LIN {X 0,Y 461.075,Z 418.748,A -85,B 0,C 180,E1 -7804.212,E2 -7804.212} C_VEL
LIN {X 0,Y 463.063,Z 429.068,A -85,B 0,C 180,E1 -7806.047,E2 -7806.047} C_VEL
LIN {X 0,Y 462.7,Z 442.277,A -85,B 0,C 180,E1 -7808.247,E2 -7808.247} C_VEL
LIN {X 0,Y 462.114,Z 460.279,A -85,B 0,C 180,E1 -7811.168,E2 -7811.168} C_VEL
LIN {X 0,Y 461.868,Z 470.776,A -85,B 0,C 180,E1 -7812.78,E2 -7812.78} C_VEL
LIN {X 0,Y 464.544,Z 487.091,A -85,B 0,C 180,E1 -7813.146,E2 -7813.146} C_VEL
LIN {X 0,Y 463.76,Z 579.084,A -85,B 0,C 180,E1 -7814.593,E2 -7814.593} C_VEL
LIN {X 0,Y 463.497,Z 592.115,A -85,B 0,C 180,E1 -7814.95,E2 -7814.95} C_VEL
LIN {X 0,Y 463.114,Z 604.111,A -85,B 0,C 180,E1 -7815.443,E2 -7815.443} C_VEL
LIN {X 0,Y 462.695,Z 614.977,A -85,B 0,C 180,E1 -7816.047,E2 -7816.047} C_VEL
LIN {X 0,Y 462.205,Z 627.162,A -85,B 0,C 180,E1 -7816.928,E2 -7816.928} C_VEL
LIN {X 0,Y 461.739,Z 636.874,A -85,B 0,C 180,E1 -7817.808,E2 -7817.808} C_VEL
LIN {X 0,Y 461.187,Z 645.853,A -85,B 0,C 180,E1 -7818.796,E2 -7818.796} C_VEL
LIN {X 0,Y 460.72,Z 655.499,A -85,B 0,C 180,E1 -7820.118,E2 -7820.118} C_VEL
LIN {X 0,Y 460.302,Z 663.256,A -85,B 0,C 180,E1 -7821.439,E2 -7821.439} C_VEL
LIN {X 0,Y 460.049,Z 668.5,A -85,B 0,C 180,E1 -7822.539,E2 -7822.539} C_VEL
LIN {X 0,Y 459.926,Z 673.622,A -85,B 0,C 180,E1 -7823.86,E2 -7823.86} C_VEL
LIN {X 0,Y 459.667,Z 677.595,A -85,B 0,C 180,E1 -7825.176,E2 -7825.176} C_VEL
LIN {X 0,Y 459.685,Z 680.521,A -85,B 0,C 180,E1 -7826.494,E2 -7826.494} C_VEL
LIN {X 0,Y 459.607,Z 681.946,A -85,B 0,C 180,E1 -7827.371,E2 -7827.371} C_VEL
LIN {X 0,Y 459.523,Z 683.559,A -85,B 0,C 180,E1 -7829.124,E2 -7829.124} C_VEL
LIN {X 0,Y 459.53,Z 683.796,A -85,B 0,C 180,E1 -7830,E2 -7830} C_VEL
LIN {X 0,Y 459.523,Z 683.608,A -85,B 0,C 180,E1 -7830.876,E2 -7830.876} C_VEL
LIN {X 0,Y 459.608,Z 682.058,A -85,B 0,C 180,E1 -7832.629,E2 -7832.629} C_VEL
LIN {X 0,Y 459.685,Z 680.697,A -85,B 0,C 180,E1 -7833.506,E2 -7833.506} C_VEL
LIN {X 0,Y 459.666,Z 677.835,A -85,B 0,C 180,E1 -7834.824,E2 -7834.824} C_VEL
LIN {X 0,Y 459.903,Z 673.941,A -85,B 0,C 180,E1 -7836.141,E2 -7836.141} C_VEL
LIN {X 0,Y 460.048,Z 668.901,A -85,B 0,C 180,E1 -7837.461,E2 -7837.461} C_VEL
LIN {X 0,Y 460.356,Z 662.544,A -85,B 0,C 180,E1 -7838.781,E2 -7838.781} C_VEL
LIN {X 0,Y 460.728,Z 654.648,A -85,B 0,C 180,E1 -7840.103,E2 -7840.103} C_VEL
LIN {X 0,Y 461.174,Z 646.581,A -85,B 0,C 180,E1 -7841.204,E2 -7841.204} C_VEL
LIN {X 0,Y 461.77,Z 636.675,A -85,B 0,C 180,E1 -7842.303,E2 -7842.303} C_VEL
LIN {X 0,Y 462.278,Z 625.413,A -85,B 0,C 180,E1 -7843.305,E2 -7843.305} C_VEL
LIN {X 0,Y 462.731,Z 614.667,A -85,B 0,C 180,E1 -7844.064,E2 -7844.064} C_VEL
LIN {X 0,Y 463.159,Z 602.475,A -85,B 0,C 180,E1 -7844.724,E2 -7844.724} C_VEL
LIN {X 0,Y 463.588,Z 589.016,A -85,B 0,C 180,E1 -7845.244,E2 -7845.244} C_VEL
LIN {X 0,Y 463.856,Z 576.705,A -85,B 0,C 180,E1 -7845.545,E2 -7845.545} C_VEL
LIN {X 0,Y 464.475,Z 486.012,A -85,B 0,C 180,E1 -7846.966,E2 -7846.966} C_VEL
LIN {X 0,Y 461.849,Z 470.717,A -85,B 0,C 180,E1 -7847.319,E2 -7847.319} C_VEL
LIN {X 0,Y 462.268,Z 455.006,A -85,B 0,C 180,E1 -7849.772,E2 -7849.772} C_VEL
LIN {X 0,Y 462.866,Z 438.129,A -85,B 0,C 180,E1 -7852.544,E2 -7852.544} C_VEL
LIN {X 0,Y 463.124,Z 429.695,A -85,B 0,C 180,E1 -7853.95,E2 -7853.95} C_VEL
LIN {X 0,Y 461.038,Z 418.49,A -85,B 0,C 180,E1 -7855.922,E2 -7855.922} C_VEL
LIN {X 0,Y 460.533,Z 416.122,A -85,B 0,C 180,E1 -7856.389,E2 -7856.389} C_VEL
LIN {X 0,Y 460.519,Z 416.123,A -85,B 0,C 180,E1 -7859.555,E2 -7859.555} C_VEL
LIN {X 0,Y 460.534,Z 416.119,A -85,B 0,C 180,E1 -7862.284,E2 -7862.284} C_VEL
LIN {X 0,Y 460.511,Z 416.125,A -85,B 0,C 180,E1 -7865.446,E2 -7865.446} C_VEL
LIN {X 0,Y 460.543,Z 416.118,A -85,B 0,C 180,E1 -7868.897,E2 -7868.897} C_VEL
LIN {X 0,Y 460.526,Z 416.118,A -85,B 0,C 180,E1 -7872.181,E2 -7872.181} C_VEL
LIN {X 0,Y 460.523,Z 416.122,A -85,B 0,C 180,E1 -7875.412,E2 -7875.412} C_VEL
LIN {X 0,Y 460.535,Z 416.113,A -85,B 0,C 180,E1 -7878.397,E2 -7878.397} C_VEL
LIN {X 0,Y 460.528,Z 416.118,A -85,B 0,C 180,E1 -7881.267,E2 -7881.267} C_VEL
LIN {X 0,Y 460.511,Z 416.116,A -85,B 0,C 180,E1 -7884.554,E2 -7884.554} C_VEL
LIN {X 0,Y 460.534,Z 416.116,A -85,B 0,C 180,E1 -7887.716,E2 -7887.716} C_VEL
LIN {X 0,Y 460.523,Z 416.122,A -85,B 0,C 180,E1 -7890.768,E2 -7890.768} C_VEL
LIN {X 0,Y 460.537,Z 416.17,A -85,B 0,C 180,E1 -7893.796,E2 -7893.796} C_VEL
LIN {X 0,Y 463.051,Z 429.137,A -85,B 0,C 180,E1 -7896.046,E2 -7896.046} C_VEL
LIN {X 0,Y 462.871,Z 439.211,A -85,B 0,C 180,E1 -7897.692,E2 -7897.692} C_VEL
LIN {X 0,Y 462.206,Z 460.623,A -85,B 0,C 180,E1 -7901.159,E2 -7901.159} C_VEL
LIN {X 0,Y 461.846,Z 471.213,A -85,B 0,C 180,E1 -7902.866,E2 -7902.866} C_VEL
LIN {X 0,Y 464.307,Z 486.198,A -85,B 0,C 180,E1 -7903.224,E2 -7903.224} C_VEL
LIN {X 0,Y 463.246,Z 581.333,A -85,B 0,C 180,E1 -7904.885,E2 -7904.885} C_VEL
LIN {X 0,Y 462.876,Z 595.262,A -85,B 0,C 180,E1 -7905.323,E2 -7905.323} C_VEL
LIN {X 0,Y 462.521,Z 607.291,A -85,B 0,C 180,E1 -7905.873,E2 -7905.873} C_VEL
LIN {X 0,Y 462.061,Z 619.024,A -85,B 0,C 180,E1 -7906.588,E2 -7906.588} C_VEL
LIN {X 0,Y 461.705,Z 630.854,A -85,B 0,C 180,E1 -7907.512,E2 -7907.512} C_VEL
LIN {X 0,Y 461.134,Z 641.61,A -85,B 0,C 180,E1 -7908.572,E2 -7908.572} C_VEL
LIN {X 0,Y 460.784,Z 650.701,A -85,B 0,C 180,E1 -7909.676,E2 -7909.676} C_VEL
LIN {X 0,Y 460.359,Z 659.464,A -85,B 0,C 180,E1 -7910.997,E2 -7910.997} C_VEL
LIN {X 0,Y 460.018,Z 666.532,A -85,B 0,C 180,E1 -7912.318,E2 -7912.318} C_VEL
LIN {X 0,Y 459.857,Z 671.279,A -85,B 0,C 180,E1 -7913.414,E2 -7913.414} C_VEL
LIN {X 0,Y 459.743,Z 675.889,A -85,B 0,C 180,E1 -7914.737,E2 -7914.737} C_VEL
LIN {X 0,Y 459.644,Z 678.306,A -85,B 0,C 180,E1 -7915.615,E2 -7915.615} C_VEL
LIN {X 0,Y 459.68,Z 680.256,A -85,B 0,C 180,E1 -7916.494,E2 -7916.494} C_VEL
LIN {X 0,Y 459.607,Z 681.795,A -85,B 0,C 180,E1 -7917.371,E2 -7917.371} C_VEL
LIN {X 0,Y 459.546,Z 682.865,A -85,B 0,C 180,E1 -7918.247,E2 -7918.247} C_VEL
LIN {X 0,Y 459.53,Z 683.801,A -85,B 0,C 180,E1 -7920,E2 -7920} C_VEL
LIN {X 0,Y 459.523,Z 683.624,A -85,B 0,C 180,E1 -7920.876,E2 -7920.876} C_VEL
LIN {X 0,Y 459.607,Z 682.049,A -85,B 0,C 180,E1 -7922.629,E2 -7922.629} C_VEL
LIN {X 0,Y 459.68,Z 680.61,A -85,B 0,C 180,E1 -7923.506,E2 -7923.506} C_VEL
LIN {X 0,Y 459.657,Z 677.632,A -85,B 0,C 180,E1 -7924.824,E2 -7924.824} C_VEL
LIN {X 0,Y 459.863,Z 673.568,A -85,B 0,C 180,E1 -7926.141,E2 -7926.141} C_VEL
LIN {X 0,Y 460.032,Z 667.335,A -85,B 0,C 180,E1 -7927.682,E2 -7927.682} C_VEL
LIN {X 0,Y 460.346,Z 660.433,A -85,B 0,C 180,E1 -7929.003,E2 -7929.003} C_VEL
LIN {X 0,Y 460.752,Z 651.823,A -85,B 0,C 180,E1 -7930.325,E2 -7930.325} C_VEL
LIN {X 0,Y 461.144,Z 642.972,A -85,B 0,C 180,E1 -7931.427,E2 -7931.427} C_VEL
LIN {X 0,Y 461.659,Z 632.544,A -85,B 0,C 180,E1 -7932.479,E2 -7932.479} C_VEL
LIN {X 0,Y 462.086,Z 621.018,A -85,B 0,C 180,E1 -7933.411,E2 -7933.411} C_VEL
LIN {X 0,Y 462.511,Z 608.682,A -85,B 0,C 180,E1 -7934.183,E2 -7934.183} C_VEL
LIN {X 0,Y 462.944,Z 597.112,A -85,B 0,C 180,E1 -7934.731,E2 -7934.731} C_VEL
LIN {X 0,Y 463.231,Z 583.9,A -85,B 0,C 180,E1 -7935.172,E2 -7935.172} C_VEL
LIN {X 0,Y 463.519,Z 567.35,A -85,B 0,C 180,E1 -7935.5,E2 -7935.5} C_VEL
LIN {X 0,Y 464.548,Z 486.066,A -85,B 0,C 180,E1 -7936.986,E2 -7936.986} C_VEL
LIN {X 0,Y 462.152,Z 471.916,A -85,B 0,C 180,E1 -7937.398,E2 -7937.398} C_VEL
LIN {X 0,Y 462.715,Z 452.676,A -85,B 0,C 180,E1 -7940.447,E2 -7940.447} C_VEL
LIN {X 0,Y 463.248,Z 433.335,A -85,B 0,C 180,E1 -7943.468,E2 -7943.468} C_VEL
LIN {X 0,Y 463.221,Z 428.858,A -85,B 0,C 180,E1 -7944.183,E2 -7944.183} C_VEL
LIN {X 0,Y 461.093,Z 418.517,A -85,B 0,C 180,E1 -7945.936,E2 -7945.936} C_VEL
LIN {X 0,Y 460.518,Z 416.124,A -85,B 0,C 180,E1 -7946.36,E2 -7946.36} C_VEL
LIN {X 0,Y 460.519,Z 416.126,A -85,B 0,C 180,E1 -7949.555,E2 -7949.555} C_VEL
LIN {X 0,Y 460.533,Z 416.119,A -85,B 0,C 180,E1 -7952.284,E2 -7952.284} C_VEL
LIN {X 0,Y 460.511,Z 416.125,A -85,B 0,C 180,E1 -7955.446,E2 -7955.446} C_VEL
LIN {X 0,Y 460.546,Z 416.118,A -85,B 0,C 180,E1 -7958.897,E2 -7958.897} C_VEL
LIN {X 0,Y 460.525,Z 416.118,A -85,B 0,C 180,E1 -7962.181,E2 -7962.181} C_VEL
LIN {X 0,Y 460.52,Z 416.122,A -85,B 0,C 180,E1 -7965.411,E2 -7965.411} C_VEL
LIN {X 0,Y 460.534,Z 416.12,A -85,B 0,C 180,E1 -7968.397,E2 -7968.397} C_VEL
LIN {X 0,Y 460.527,Z 416.119,A -85,B 0,C 180,E1 -7971.267,E2 -7971.267} C_VEL
LIN {X 0,Y 460.511,Z 416.122,A -85,B 0,C 180,E1 -7974.554,E2 -7974.554} C_VEL
LIN {X 0,Y 460.533,Z 416.118,A -85,B 0,C 180,E1 -7977.716,E2 -7977.716} C_VEL
LIN {X 0,Y 460.546,Z 416.195,A -85,B 0,C 180,E1 -7981.019,E2 -7981.019} C_VEL
LIN {X 0,Y 463.789,Z 431.549,A -85,B 0,C 180,E1 -7983.587,E2 -7983.587} C_VEL
LIN {X 0,Y 463.673,Z 438.411,A -85,B 0,C 180,E1 -7984.647,E2 -7984.647} C_VEL
LIN {X 0,Y 462.791,Z 458.476,A -85,B 0,C 180,E1 -7987.688,E2 -7987.688} C_VEL
LIN {X 0,Y 461.825,Z 481.82,A -85,B 0,C 180,E1 -7991.173,E2 -7991.173} C_VEL
LIN {X 0,Y 461.381,Z 492.48,A -85,B 0,C 180,E1 -7992.75,E2 -7992.75} C_VEL
LIN {X 0,Y 464.124,Z 514.756,A -85,B 0,C 180,E1 -7993.251,E2 -7993.251} C_VEL
LIN {X 0,Y 463.33,Z 592.644,A -85,B 0,C 180,E1 -7994.578,E2 -7994.578} C_VEL
LIN {X 0,Y 463.11,Z 609.106,A -85,B 0,C 180,E1 -7994.881,E2 -7994.881} C_VEL
LIN {X 0,Y 462.775,Z 621.21,A -85,B 0,C 180,E1 -7995.263,E2 -7995.263} C_VEL
LIN {X 0,Y 462.308,Z 633.167,A -85,B 0,C 180,E1 -7995.81,E2 -7995.81} C_VEL
LIN {X 0,Y 461.887,Z 645.584,A -85,B 0,C 180,E1 -7996.583,E2 -7996.583} C_VEL
LIN {X 0,Y 461.421,Z 656.045,A -85,B 0,C 180,E1 -7997.412,E2 -7997.412} C_VEL
LIN {X 0,Y 460.979,Z 665.561,A -85,B 0,C 180,E1 -7998.346,E2 -7998.346} C_VEL
LIN {X 0,Y 460.53,Z 674.702,A -85,B 0,C 180,E1 -7999.448,E2 -7999.448} C_VEL
LIN {X 0,Y 460.165,Z 683.581,A -85,B 0,C 180,E1 -8000.772,E2 -8000.772} C_VEL
LIN {X 0,Y 459.921,Z 690.697,A -85,B 0,C 180,E1 -8002.095,E2 -8002.095} C_VEL
LIN {X 0,Y 459.719,Z 696.887,A -85,B 0,C 180,E1 -8003.564,E2 -8003.564} C_VEL
LIN {X 0,Y 459.652,Z 702.015,A -85,B 0,C 180,E1 -8005.176,E2 -8005.176} C_VEL
LIN {X 0,Y 459.697,Z 704.999,A -85,B 0,C 180,E1 -8006.494,E2 -8006.494} C_VEL
LIN {X 0,Y 459.64,Z 706.431,A -85,B 0,C 180,E1 -8007.371,E2 -8007.371} C_VEL
LIN {X 0,Y 459.596,Z 708.057,A -85,B 0,C 180,E1 -8009.124,E2 -8009.124} C_VEL
LIN {X 0,Y 459.584,Z 708.278,A -85,B 0,C 180,E1 -8010,E2 -8010} C_VEL
LIN {X 0,Y 459.596,Z 708.057,A -85,B 0,C 180,E1 -8010.876,E2 -8010.876} C_VEL
LIN {X 0,Y 459.642,Z 706.431,A -85,B 0,C 180,E1 -8012.629,E2 -8012.629} C_VEL
LIN {X 0,Y 459.708,Z 705,A -85,B 0,C 180,E1 -8013.506,E2 -8013.506} C_VEL
LIN {X 0,Y 459.66,Z 702.015,A -85,B 0,C 180,E1 -8014.824,E2 -8014.824} C_VEL
LIN {X 0,Y 459.765,Z 696.7,A -85,B 0,C 180,E1 -8016.487,E2 -8016.487} C_VEL
LIN {X 0,Y 459.925,Z 690.699,A -85,B 0,C 180,E1 -8017.905,E2 -8017.905} C_VEL
LIN {X 0,Y 460.19,Z 683.584,A -85,B 0,C 180,E1 -8019.228,E2 -8019.228} C_VEL
LIN {X 0,Y 460.54,Z 674.691,A -85,B 0,C 180,E1 -8020.552,E2 -8020.552} C_VEL
LIN {X 0,Y 460.979,Z 665.542,A -85,B 0,C 180,E1 -8021.654,E2 -8021.654} C_VEL
LIN {X 0,Y 461.492,Z 655.22,A -85,B 0,C 180,E1 -8022.656,E2 -8022.656} C_VEL
LIN {X 0,Y 461.929,Z 643.989,A -85,B 0,C 180,E1 -8023.528,E2 -8023.528} C_VEL
LIN {X 0,Y 462.4,Z 632.124,A -85,B 0,C 180,E1 -8024.243,E2 -8024.243} C_VEL
LIN {X 0,Y 462.835,Z 619.661,A -85,B 0,C 180,E1 -8024.791,E2 -8024.791} C_VEL
LIN {X 0,Y 463.161,Z 606.804,A -85,B 0,C 180,E1 -8025.174,E2 -8025.174} C_VEL
LIN {X 0,Y 463.762,Z 546.734,A -85,B 0,C 180,E1 -8026.193,E2 -8026.193} C_VEL
LIN {X 0,Y 464.092,Z 513.352,A -85,B 0,C 180,E1 -8026.813,E2 -8026.813} C_VEL
LIN {X 0,Y 461.241,Z 488.658,A -85,B 0,C 180,E1 -8027.437,E2 -8027.437} C_VEL
LIN {X 0,Y 462.12,Z 465.23,A -85,B 0,C 180,E1 -8030.94,E2 -8030.94} C_VEL
LIN {X 0,Y 463.02,Z 444.03,A -85,B 0,C 180,E1 -8034.194,E2 -8034.194} C_VEL
LIN {X 0,Y 463.674,Z 432.077,A -85,B 0,C 180,E1 -8036.076,E2 -8036.076} C_VEL
LIN {X 0,Y 462.51,Z 424.778,A -85,B 0,C 180,E1 -8037.341,E2 -8037.341} C_VEL
LIN {X 0,Y 460.541,Z 416.122,A -85,B 0,C 180,E1 -8038.981,E2 -8038.981} C_VEL
LIN {X 0,Y 460.533,Z 416.12,A -85,B 0,C 180,E1 -8042.284,E2 -8042.284} C_VEL
LIN {X 0,Y 460.51,Z 416.125,A -85,B 0,C 180,E1 -8045.446,E2 -8045.446} C_VEL
LIN {X 0,Y 460.534,Z 416.119,A -85,B 0,C 180,E1 -8048.896,E2 -8048.896} C_VEL
LIN {X 0,Y 460.52,Z 416.122,A -85,B 0,C 180,E1 -8051.601,E2 -8051.601} C_VEL
LIN {X 0,Y 460.518,Z 416.12,A -85,B 0,C 180,E1 -8054.589,E2 -8054.589} C_VEL
LIN {X 0,Y 460.525,Z 416.118,A -85,B 0,C 180,E1 -8057.819,E2 -8057.819} C_VEL
LIN {X 0,Y 460.547,Z 416.119,A -85,B 0,C 180,E1 -8061.102,E2 -8061.102} C_VEL
LIN {X 0,Y 460.513,Z 416.121,A -85,B 0,C 180,E1 -8064.554,E2 -8064.554} C_VEL
LIN {X 0,Y 460.534,Z 416.118,A -85,B 0,C 180,E1 -8067.716,E2 -8067.716} C_VEL
LIN {X 0,Y 460.542,Z 416.121,A -85,B 0,C 180,E1 -8070.769,E2 -8070.769} C_VEL
LIN {X 0,Y 460.559,Z 416.116,A -85,B 0,C 180,E1 -8073.734,E2 -8073.734} C_VEL
LIN {X 0,Y 460.547,Z 416.123,A -85,B 0,C 180,E1 -8076.624,E2 -8076.624} C_VEL
LIN {X 0,Y 460.553,Z 416.117,A -85,B 0,C 180,E1 -8079.453,E2 -8079.453} C_VEL
LIN {X 0,Y 460.568,Z 416.117,A -85,B 0,C 180,E1 -8082.643,E2 -8082.643} C_VEL
LIN {X 0,Y 460.578,Z 416.182,A -85,B 0,C 180,E1 -8082.713,E2 -8082.713} C_VEL
LIN {X 0,Y 462.882,Z 422.42,A -85,B 0,C 180,E1 -8082.954,E2 -8082.954} C_VEL
LIN {X 0,Y 464.811,Z 427.449,A -85,B 0,C 180,E1 -8083.149,E2 -8083.149} C_VEL
LIN {X 0,Y 463.534,Z 519.172,A -85,B 0,C 180,E1 -8084.867,E2 -8084.867} C_VEL
LIN {X 0,Y 463.331,Z 532.093,A -85,B 0,C 180,E1 -8085.281,E2 -8085.281} C_VEL
LIN {X 0,Y 463.084,Z 544.075,A -85,B 0,C 180,E1 -8085.835,E2 -8085.835} C_VEL
LIN {X 0,Y 462.679,Z 555.95,A -85,B 0,C 180,E1 -8086.568,E2 -8086.568} C_VEL
LIN {X 0,Y 462.241,Z 567.55,A -85,B 0,C 180,E1 -8087.487,E2 -8087.487} C_VEL
LIN {X 0,Y 461.85,Z 576.525,A -85,B 0,C 180,E1 -8088.368,E2 -8088.368} C_VEL
LIN {X 0,Y 461.424,Z 585.721,A -85,B 0,C 180,E1 -8089.469,E2 -8089.469} C_VEL
LIN {X 0,Y 460.993,Z 594.604,A -85,B 0,C 180,E1 -8090.789,E2 -8090.789} C_VEL
LIN {X 0,Y 460.65,Z 601.715,A -85,B 0,C 180,E1 -8092.108,E2 -8092.108} C_VEL
LIN {X 0,Y 460.422,Z 607.329,A -85,B 0,C 180,E1 -8093.426,E2 -8093.426} C_VEL
LIN {X 0,Y 460.148,Z 611.72,A -85,B 0,C 180,E1 -8094.742,E2 -8094.742} C_VEL
LIN {X 0,Y 460.171,Z 614,A -85,B 0,C 180,E1 -8095.62,E2 -8095.62} C_VEL
LIN {X 0,Y 459.993,Z 615.87,A -85,B 0,C 180,E1 -8096.496,E2 -8096.496} C_VEL
LIN {X 0,Y 459.819,Z 617.29,A -85,B 0,C 180,E1 -8097.372,E2 -8097.372} C_VEL
LIN {X 0,Y 459.691,Z 618.83,A -85,B 0,C 180,E1 -8099.124,E2 -8099.124} C_VEL
LIN {X 0,Y 459.679,Z 619.005,A -85,B 0,C 180,E1 -8100,E2 -8100} C_VEL
LIN {X 0,Y 459.679,Z 618.737,A -85,B 0,C 180,E1 -8100.876,E2 -8100.876} C_VEL
LIN {X 0,Y 459.806,Z 616.987,A -85,B 0,C 180,E1 -8102.628,E2 -8102.628} C_VEL
LIN {X 0,Y 459.987,Z 615.491,A -85,B 0,C 180,E1 -8103.504,E2 -8103.504} C_VEL
LIN {X 0,Y 460.064,Z 612.422,A -85,B 0,C 180,E1 -8104.82,E2 -8104.82} C_VEL
LIN {X 0,Y 460.201,Z 607.217,A -85,B 0,C 180,E1 -8106.421,E2 -8106.421} C_VEL
LIN {X 0,Y 460.446,Z 600.884,A -85,B 0,C 180,E1 -8107.896,E2 -8107.896} C_VEL
LIN {X 0,Y 460.798,Z 593.657,A -85,B 0,C 180,E1 -8109.215,E2 -8109.215} C_VEL
LIN {X 0,Y 461.192,Z 584.638,A -85,B 0,C 180,E1 -8110.537,E2 -8110.537} C_VEL
LIN {X 0,Y 461.645,Z 575.368,A -85,B 0,C 180,E1 -8111.637,E2 -8111.637} C_VEL
LIN {X 0,Y 462.056,Z 565.037,A -85,B 0,C 180,E1 -8112.63,E2 -8112.63} C_VEL
LIN {X 0,Y 462.46,Z 553.768,A -85,B 0,C 180,E1 -8113.499,E2 -8113.499} C_VEL
LIN {X 0,Y 462.783,Z 541.687,A -85,B 0,C 180,E1 -8114.231,E2 -8114.231} C_VEL
LIN {X 0,Y 463.115,Z 528.597,A -85,B 0,C 180,E1 -8114.81,E2 -8114.81} C_VEL
LIN {X 0,Y 463.364,Z 515.877,A -85,B 0,C 180,E1 -8115.195,E2 -8115.195} C_VEL
LIN {X 0,Y 464.244,Z 426.98,A -85,B 0,C 180,E1 -8116.76,E2 -8116.76} C_VEL
LIN {X 0,Y 460.544,Z 416.12,A -85,B 0,C 180,E1 -8117.112,E2 -8117.112} C_VEL
LIN {X 0,Y 460.569,Z 416.121,A -85,B 0,C 180,E1 -8119.616,E2 -8119.616} C_VEL
LIN {X 0,Y 460.513,Z 416.117,A -85,B 0,C 180,E1 -8122.429,E2 -8122.429} C_VEL
LIN {X 0,Y 460.548,Z 416.115,A -85,B 0,C 180,E1 -8125.796,E2 -8125.796} C_VEL
LIN {X 0,Y 460.552,Z 416.11,A -85,B 0,C 180,E1 -8128.233,E2 -8128.233} C_VEL
LIN {X 0,Y 460.524,Z 416.118,A -85,B 0,C 180,E1 -8131.283,E2 -8131.283} C_VEL
LIN {X 0,Y 460.534,Z 416.105,A -85,B 0,C 180,E1 -8134.505,E2 -8134.505} C_VEL
LIN {X 0,Y 460.504,Z 416.122,A -85,B 0,C 180,E1 -8137.623,E2 -8137.623} C_VEL
LIN {X 0,Y 460.542,Z 416.109,A -85,B 0,C 180,E1 -8140.269,E2 -8140.269} C_VEL
LIN {X 0,Y 460.503,Z 416.123,A -85,B 0,C 180,E1 -8143.375,E2 -8143.375} C_VEL
LIN {X 0,Y 460.503,Z 416.118,A -85,B 0,C 180,E1 -8146.625,E2 -8146.625} C_VEL
LIN {X 0,Y 460.542,Z 416.11,A -85,B 0,C 180,E1 -8149.731,E2 -8149.731} C_VEL
LIN {X 0,Y 460.499,Z 416.124,A -85,B 0,C 180,E1 -8152.524,E2 -8152.524} C_VEL
LIN {X 0,Y 460.548,Z 416.114,A -85,B 0,C 180,E1 -8155.624,E2 -8155.624} C_VEL
LIN {X 0,Y 460.54,Z 416.122,A -85,B 0,C 180,E1 -8158.745,E2 -8158.745} C_VEL
LIN {X 0,Y 460.51,Z 416.125,A -85,B 0,C 180,E1 -8161.764,E2 -8161.764} C_VEL
LIN {X 0,Y 460.555,Z 416.234,A -85,B 0,C 180,E1 -8163.765,E2 -8163.765} C_VEL
LIN {X 0,Y 461.075,Z 418.748,A -85,B 0,C 180,E1 -8164.212,E2 -8164.212} C_VEL
LIN {X 0,Y 461.098,Z 422.256,A -85,B 0,C 180,E1 -8164.803,E2 -8164.803} C_VEL
LIN {X 0,Y 460.118,Z 425.937,A -85,B 0,C 180,E1 -8165.373,E2 -8165.373} C_VEL
LIN {X 0,Y 456.381,Z 435.933,A -85,B 0,C 180,E1 -8166.877,E2 -8166.877} C_VEL
LIN {X 0,Y 455.999,Z 438.386,A -85,B 0,C 180,E1 -8167.274,E2 -8167.274} C_VEL
LIN {X 0,Y 455.271,Z 457.786,A -85,B 0,C 180,E1 -8170.476,E2 -8170.476} C_VEL
LIN {X 0,Y 454.939,Z 470.902,A -85,B 0,C 180,E1 -8172.51,E2 -8172.51} C_VEL
LIN {X 0,Y 457.737,Z 487.036,A -85,B 0,C 180,E1 -8172.885,E2 -8172.885} C_VEL
LIN {X 0,Y 456.936,Z 579.198,A -85,B 0,C 180,E1 -8174.357,E2 -8174.357} C_VEL
LIN {X 0,Y 456.665,Z 592.262,A -85,B 0,C 180,E1 -8174.719,E2 -8174.719} C_VEL
LIN {X 0,Y 456.271,Z 604.275,A -85,B 0,C 180,E1 -8175.22,E2 -8175.22} C_VEL
LIN {X 0,Y 455.814,Z 615.149,A -85,B 0,C 180,E1 -8175.832,E2 -8175.832} C_VEL
LIN {X 0,Y 455.286,Z 627.235,A -85,B 0,C 180,E1 -8176.717,E2 -8176.717} C_VEL
LIN {X 0,Y 454.82,Z 637.055,A -85,B 0,C 180,E1 -8177.62,E2 -8177.62} C_VEL
LIN {X 0,Y 454.232,Z 646.036,A -85,B 0,C 180,E1 -8178.623,E2 -8178.623} C_VEL
LIN {X 0,Y 453.768,Z 654.242,A -85,B 0,C 180,E1 -8179.74,E2 -8179.74} C_VEL
LIN {X 0,Y 453.355,Z 662.245,A -85,B 0,C 180,E1 -8181.082,E2 -8181.082} C_VEL
LIN {X 0,Y 452.992,Z 668.688,A -85,B 0,C 180,E1 -8182.422,E2 -8182.422} C_VEL
LIN {X 0,Y 452.856,Z 673.811,A -85,B 0,C 180,E1 -8183.763,E2 -8183.763} C_VEL
LIN {X 0,Y 452.6,Z 677.784,A -85,B 0,C 180,E1 -8185.101,E2 -8185.101} C_VEL
LIN {X 0,Y 452.601,Z 680.711,A -85,B 0,C 180,E1 -8186.439,E2 -8186.439} C_VEL
LIN {X 0,Y 452.534,Z 682.135,A -85,B 0,C 180,E1 -8187.33,E2 -8187.33} C_VEL
LIN {X 0,Y 452.43,Z 683.748,A -85,B 0,C 180,E1 -8189.11,E2 -8189.11} C_VEL
LIN {X 0,Y 452.435,Z 683.985,A -85,B 0,C 180,E1 -8190,E2 -8190} C_VEL
LIN {X 0,Y 452.43,Z 683.796,A -85,B 0,C 180,E1 -8190.89,E2 -8190.89} C_VEL
LIN {X 0,Y 452.534,Z 682.246,A -85,B 0,C 180,E1 -8192.67,E2 -8192.67} C_VEL
LIN {X 0,Y 452.601,Z 680.884,A -85,B 0,C 180,E1 -8193.561,E2 -8193.561} C_VEL
LIN {X 0,Y 452.599,Z 678.022,A -85,B 0,C 180,E1 -8194.899,E2 -8194.899} C_VEL
LIN {X 0,Y 452.831,Z 674.127,A -85,B 0,C 180,E1 -8196.237,E2 -8196.237} C_VEL
LIN {X 0,Y 452.991,Z 669.086,A -85,B 0,C 180,E1 -8197.578,E2 -8197.578} C_VEL
LIN {X 0,Y 453.34,Z 662.726,A -85,B 0,C 180,E1 -8198.918,E2 -8198.918} C_VEL
LIN {X 0,Y 453.739,Z 654.828,A -85,B 0,C 180,E1 -8200.261,E2 -8200.261} C_VEL
LIN {X 0,Y 454.21,Z 646.758,A -85,B 0,C 180,E1 -8201.378,E2 -8201.378} C_VEL
LIN {X 0,Y 454.835,Z 636.848,A -85,B 0,C 180,E1 -8202.493,E2 -8202.493} C_VEL
LIN {X 0,Y 455.346,Z 625.724,A -85,B 0,C 180,E1 -8203.499,E2 -8203.499} C_VEL
LIN {X 0,Y 455.851,Z 614.825,A -85,B 0,C 180,E1 -8204.281,E2 -8204.281} C_VEL
LIN {X 0,Y 456.318,Z 602.616,A -85,B 0,C 180,E1 -8204.95,E2 -8204.95} C_VEL
LIN {X 0,Y 456.761,Z 589.133,A -85,B 0,C 180,E1 -8205.478,E2 -8205.478} C_VEL
LIN {X 0,Y 457.046,Z 576.746,A -85,B 0,C 180,E1 -8205.782,E2 -8205.782} C_VEL
LIN {X 0,Y 457.62,Z 486.269,A -85,B 0,C 180,E1 -8207.224,E2 -8207.224} C_VEL
LIN {X 0,Y 454.952,Z 470.855,A -85,B 0,C 180,E1 -8207.587,E2 -8207.587} C_VEL
LIN {X 0,Y 455.382,Z 454.985,A -85,B 0,C 180,E1 -8210.084,E2 -8210.084} C_VEL
LIN {X 0,Y 456.034,Z 437.992,A -85,B 0,C 180,E1 -8212.901,E2 -8212.901} C_VEL
LIN {X 0,Y 456.194,Z 430.883,A -85,B 0,C 180,E1 -8214.091,E2 -8214.091} C_VEL
LIN {X 0,Y 453.772,Z 418.331,A -85,B 0,C 180,E1 -8216.336,E2 -8216.336} C_VEL
LIN {X 0,Y 453.472,Z 417.002,A -85,B 0,C 180,E1 -8216.62,E2 -8216.62} C_VEL
LIN {X 0,Y 453.471,Z 417.001,A -85,B 0,C 180,E1 -8219.784,E2 -8219.784} C_VEL
LIN {X 0,Y 453.493,Z 416.998,A -85,B 0,C 180,E1 -8223.189,E2 -8223.189} C_VEL
LIN {X 0,Y 453.453,Z 417.001,A -85,B 0,C 180,E1 -8226.298,E2 -8226.298} C_VEL
LIN {X 0,Y 453.488,Z 416.995,A -85,B 0,C 180,E1 -8229.45,E2 -8229.45} C_VEL
LIN {X 0,Y 453.479,Z 416.996,A -85,B 0,C 180,E1 -8231.935,E2 -8231.935} C_VEL
LIN {X 0,Y 453.494,Z 416.997,A -85,B 0,C 180,E1 -8235.47,E2 -8235.47} C_VEL
LIN {X 0,Y 453.482,Z 416.991,A -85,B 0,C 180,E1 -8238.209,E2 -8238.209} C_VEL
LIN {X 0,Y 453.512,Z 416.998,A -85,B 0,C 180,E1 -8240.791,E2 -8240.791} C_VEL
LIN {X 0,Y 453.454,Z 416.989,A -85,B 0,C 180,E1 -8243.917,E2 -8243.917} C_VEL
LIN {X 0,Y 453.486,Z 416.996,A -85,B 0,C 180,E1 -8247.151,E2 -8247.151} C_VEL
LIN {X 0,Y 453.465,Z 417.002,A -85,B 0,C 180,E1 -8250.267,E2 -8250.267} C_VEL
LIN {X 0,Y 453.492,Z 416.996,A -85,B 0,C 180,E1 -8253.574,E2 -8253.574} C_VEL
LIN {X 0,Y 456.116,Z 430.323,A -85,B 0,C 180,E1 -8255.92,E2 -8255.92} C_VEL
LIN {X 0,Y 456.042,Z 438.922,A -85,B 0,C 180,E1 -8257.339,E2 -8257.339} C_VEL
LIN {X 0,Y 455.275,Z 460.69,A -85,B 0,C 180,E1 -8260.89,E2 -8260.89} C_VEL
LIN {X 0,Y 454.879,Z 471.285,A -85,B 0,C 180,E1 -8262.614,E2 -8262.614} C_VEL
LIN {X 0,Y 457.419,Z 486.804,A -85,B 0,C 180,E1 -8262.997,E2 -8262.997} C_VEL
LIN {X 0,Y 456.349,Z 580.94,A -85,B 0,C 180,E1 -8264.68,E2 -8264.68} C_VEL
LIN {X 0,Y 455.963,Z 594.3,A -85,B 0,C 180,E1 -8265.095,E2 -8265.095} C_VEL
LIN {X 0,Y 455.613,Z 606.644,A -85,B 0,C 180,E1 -8265.654,E2 -8265.654} C_VEL
LIN {X 0,Y 455.112,Z 618.568,A -85,B 0,C 180,E1 -8266.379,E2 -8266.379} C_VEL
LIN {X 0,Y 454.817,Z 628.793,A -85,B 0,C 180,E1 -8267.169,E2 -8267.169} C_VEL
LIN {X 0,Y 454.284,Z 639.377,A -85,B 0,C 180,E1 -8268.171,E2 -8268.171} C_VEL
LIN {X 0,Y 453.787,Z 648.868,A -85,B 0,C 180,E1 -8269.289,E2 -8269.289} C_VEL
LIN {X 0,Y 453.352,Z 658.109,A -85,B 0,C 180,E1 -8270.632,E2 -8270.632} C_VEL
LIN {X 0,Y 453.022,Z 665.453,A -85,B 0,C 180,E1 -8271.974,E2 -8271.974} C_VEL
LIN {X 0,Y 452.769,Z 671.8,A -85,B 0,C 180,E1 -8273.428,E2 -8273.428} C_VEL
LIN {X 0,Y 452.688,Z 675.981,A -85,B 0,C 180,E1 -8274.655,E2 -8274.655} C_VEL
LIN {X 0,Y 452.558,Z 678.427,A -85,B 0,C 180,E1 -8275.547,E2 -8275.547} C_VEL
LIN {X 0,Y 452.581,Z 680.393,A -85,B 0,C 180,E1 -8276.439,E2 -8276.439} C_VEL
LIN {X 0,Y 452.533,Z 681.947,A -85,B 0,C 180,E1 -8277.33,E2 -8277.33} C_VEL
LIN {X 0,Y 452.461,Z 683.036,A -85,B 0,C 180,E1 -8278.22,E2 -8278.22} C_VEL
LIN {X 0,Y 452.435,Z 683.991,A -85,B 0,C 180,E1 -8280,E2 -8280} C_VEL
LIN {X 0,Y 452.43,Z 683.826,A -85,B 0,C 180,E1 -8280.89,E2 -8280.89} C_VEL
LIN {X 0,Y 452.461,Z 683.241,A -85,B 0,C 180,E1 -8281.78,E2 -8281.78} C_VEL
LIN {X 0,Y 452.533,Z 682.259,A -85,B 0,C 180,E1 -8282.67,E2 -8282.67} C_VEL
LIN {X 0,Y 452.596,Z 680.827,A -85,B 0,C 180,E1 -8283.561,E2 -8283.561} C_VEL
LIN {X 0,Y 452.591,Z 677.847,A -85,B 0,C 180,E1 -8284.899,E2 -8284.899} C_VEL
LIN {X 0,Y 452.792,Z 673.779,A -85,B 0,C 180,E1 -8286.238,E2 -8286.238} C_VEL
LIN {X 0,Y 452.995,Z 667.544,A -85,B 0,C 180,E1 -8287.802,E2 -8287.802} C_VEL
LIN {X 0,Y 453.334,Z 660.639,A -85,B 0,C 180,E1 -8289.143,E2 -8289.143} C_VEL
LIN {X 0,Y 453.768,Z 652.028,A -85,B 0,C 180,E1 -8290.485,E2 -8290.485} C_VEL
LIN {X 0,Y 454.188,Z 643.159,A -85,B 0,C 180,E1 -8291.605,E2 -8291.605} C_VEL
LIN {X 0,Y 454.712,Z 632.916,A -85,B 0,C 180,E1 -8292.656,E2 -8292.656} C_VEL
LIN {X 0,Y 455.145,Z 622.743,A -85,B 0,C 180,E1 -8293.506,E2 -8293.506} C_VEL
LIN {X 0,Y 455.565,Z 610.878,A -85,B 0,C 180,E1 -8294.29,E2 -8294.29} C_VEL
LIN {X 0,Y 456.02,Z 598.658,A -85,B 0,C 180,E1 -8294.903,E2 -8294.903} C_VEL
LIN {X 0,Y 456.353,Z 586.282,A -85,B 0,C 180,E1 -8295.349,E2 -8295.349} C_VEL
LIN {X 0,Y 456.663,Z 571.158,A -85,B 0,C 180,E1 -8295.681,E2 -8295.681} C_VEL
LIN {X 0,Y 457.931,Z 487.484,A -85,B 0,C 180,E1 -8297.254,E2 -8297.254} C_VEL
LIN {X 0,Y 455.317,Z 472.331,A -85,B 0,C 180,E1 -8297.691,E2 -8297.691} C_VEL
LIN {X 0,Y 455.897,Z 453.053,A -85,B 0,C 180,E1 -8300.767,E2 -8300.767} C_VEL
LIN {X 0,Y 456.456,Z 435.128,A -85,B 0,C 180,E1 -8303.598,E2 -8303.598} C_VEL
LIN {X 0,Y 456.35,Z 430.149,A -85,B 0,C 180,E1 -8304.405,E2 -8304.405} C_VEL
LIN {X 0,Y 454.003,Z 419.118,A -85,B 0,C 180,E1 -8306.324,E2 -8306.324} C_VEL
LIN {X 0,Y 453.477,Z 417,A -85,B 0,C 180,E1 -8306.708,E2 -8306.708} C_VEL
LIN {X 0,Y 453.47,Z 417.004,A -85,B 0,C 180,E1 -8309.784,E2 -8309.784} C_VEL
LIN {X 0,Y 453.493,Z 417,A -85,B 0,C 180,E1 -8313.189,E2 -8313.189} C_VEL
LIN {X 0,Y 453.452,Z 416.999,A -85,B 0,C 180,E1 -8316.298,E2 -8316.298} C_VEL
LIN {X 0,Y 453.492,Z 416.996,A -85,B 0,C 180,E1 -8319.45,E2 -8319.45} C_VEL
LIN {X 0,Y 453.479,Z 416.997,A -85,B 0,C 180,E1 -8321.935,E2 -8321.935} C_VEL
LIN {X 0,Y 453.49,Z 416.998,A -85,B 0,C 180,E1 -8325.471,E2 -8325.471} C_VEL
LIN {X 0,Y 453.481,Z 416.997,A -85,B 0,C 180,E1 -8328.209,E2 -8328.209} C_VEL
LIN {X 0,Y 453.496,Z 416.995,A -85,B 0,C 180,E1 -8330.793,E2 -8330.793} C_VEL
LIN {X 0,Y 453.453,Z 416.999,A -85,B 0,C 180,E1 -8333.917,E2 -8333.917} C_VEL
LIN {X 0,Y 453.485,Z 416.997,A -85,B 0,C 180,E1 -8337.151,E2 -8337.151} C_VEL
LIN {X 0,Y 453.513,Z 416.997,A -85,B 0,C 180,E1 -8340.781,E2 -8340.781} C_VEL
LIN {X 0,Y 456.87,Z 433.019,A -85,B 0,C 180,E1 -8343.506,E2 -8343.506} C_VEL
LIN {X 0,Y 456.522,Z 445.458,A -85,B 0,C 180,E1 -8345.439,E2 -8345.439} C_VEL
LIN {X 0,Y 455.514,Z 465.486,A -85,B 0,C 180,E1 -8348.504,E2 -8348.504} C_VEL
LIN {X 0,Y 454.546,Z 488.512,A -85,B 0,C 180,E1 -8351.987,E2 -8351.987} C_VEL
LIN {X 0,Y 454.401,Z 491.955,A -85,B 0,C 180,E1 -8352.505,E2 -8352.505} C_VEL
LIN {X 0,Y 457.276,Z 516.196,A -85,B 0,C 180,E1 -8353.051,E2 -8353.051} C_VEL
LIN {X 0,Y 456.674,Z 569.237,A -85,B 0,C 180,E1 -8353.975,E2 -8353.975} C_VEL
LIN {X 0,Y 456.26,Z 606.763,A -85,B 0,C 180,E1 -8354.591,E2 -8354.591} C_VEL
LIN {X 0,Y 455.946,Z 620.322,A -85,B 0,C 180,E1 -8355.009,E2 -8355.009} C_VEL
LIN {X 0,Y 455.413,Z 633.01,A -85,B 0,C 180,E1 -8355.591,E2 -8355.591} C_VEL
LIN {X 0,Y 454.966,Z 645.418,A -85,B 0,C 180,E1 -8356.375,E2 -8356.375} C_VEL
LIN {X 0,Y 454.447,Z 656.302,A -85,B 0,C 180,E1 -8357.254,E2 -8357.254} C_VEL
LIN {X 0,Y 453.949,Z 665.383,A -85,B 0,C 180,E1 -8358.163,E2 -8358.163} C_VEL
LIN {X 0,Y 453.525,Z 674.521,A -85,B 0,C 180,E1 -8359.283,E2 -8359.283} C_VEL
LIN {X 0,Y 453.134,Z 683.398,A -85,B 0,C 180,E1 -8360.627,E2 -8360.627} C_VEL
LIN {X 0,Y 452.856,Z 690.511,A -85,B 0,C 180,E1 -8361.971,E2 -8361.971} C_VEL
LIN {X 0,Y 452.63,Z 697.132,A -85,B 0,C 180,E1 -8363.582,E2 -8363.582} C_VEL
LIN {X 0,Y 452.579,Z 701.828,A -85,B 0,C 180,E1 -8365.1,E2 -8365.1} C_VEL
LIN {X 0,Y 452.59,Z 704.811,A -85,B 0,C 180,E1 -8366.439,E2 -8366.439} C_VEL
LIN {X 0,Y 452.564,Z 706.243,A -85,B 0,C 180,E1 -8367.33,E2 -8367.33} C_VEL
LIN {X 0,Y 452.499,Z 707.868,A -85,B 0,C 180,E1 -8369.11,E2 -8369.11} C_VEL
LIN {X 0,Y 452.515,Z 708.09,A -85,B 0,C 180,E1 -8370,E2 -8370} C_VEL
LIN {X 0,Y 452.499,Z 707.868,A -85,B 0,C 180,E1 -8370.89,E2 -8370.89} C_VEL
LIN {X 0,Y 452.566,Z 706.243,A -85,B 0,C 180,E1 -8372.67,E2 -8372.67} C_VEL
LIN {X 0,Y 452.601,Z 704.811,A -85,B 0,C 180,E1 -8373.561,E2 -8373.561} C_VEL
LIN {X 0,Y 452.586,Z 701.827,A -85,B 0,C 180,E1 -8374.899,E2 -8374.899} C_VEL
LIN {X 0,Y 452.691,Z 696.883,A -85,B 0,C 180,E1 -8376.486,E2 -8376.486} C_VEL
LIN {X 0,Y 452.86,Z 690.511,A -85,B 0,C 180,E1 -8378.029,E2 -8378.029} C_VEL
LIN {X 0,Y 453.156,Z 683.399,A -85,B 0,C 180,E1 -8379.372,E2 -8379.372} C_VEL
LIN {X 0,Y 453.529,Z 674.507,A -85,B 0,C 180,E1 -8380.717,E2 -8380.717} C_VEL
LIN {X 0,Y 453.982,Z 665.36,A -85,B 0,C 180,E1 -8381.837,E2 -8381.837} C_VEL
LIN {X 0,Y 454.537,Z 654.905,A -85,B 0,C 180,E1 -8382.865,E2 -8382.865} C_VEL
LIN {X 0,Y 455.007,Z 643.816,A -85,B 0,C 180,E1 -8383.738,E2 -8383.738} C_VEL
LIN {X 0,Y 455.501,Z 631.96,A -85,B 0,C 180,E1 -8384.463,E2 -8384.463} C_VEL
LIN {X 0,Y 455.977,Z 618.759,A -85,B 0,C 180,E1 -8385.047,E2 -8385.047} C_VEL
LIN {X 0,Y 456.382,Z 605.545,A -85,B 0,C 180,E1 -8385.434,E2 -8385.434} C_VEL
LIN {X 0,Y 456.924,Z 555.768,A -85,B 0,C 180,E1 -8386.277,E2 -8386.277} C_VEL
LIN {X 0,Y 457.332,Z 513.967,A -85,B 0,C 180,E1 -8387.077,E2 -8387.077} C_VEL
LIN {X 0,Y 454.25,Z 487.841,A -85,B 0,C 180,E1 -8387.753,E2 -8387.753} C_VEL
LIN {X 0,Y 455.139,Z 466.283,A -85,B 0,C 180,E1 -8391.04,E2 -8391.04} C_VEL
LIN {X 0,Y 456.133,Z 445.223,A -85,B 0,C 180,E1 -8394.341,E2 -8394.341} C_VEL
LIN {X 0,Y 456.822,Z 433.361,A -85,B 0,C 180,E1 -8396.251,E2 -8396.251} C_VEL
LIN {X 0,Y 455.035,Z 423.426,A -85,B 0,C 180,E1 -8398.053,E2 -8398.053} C_VEL
LIN {X 0,Y 453.478,Z 417.004,A -85,B 0,C 180,E1 -8399.317,E2 -8399.317} C_VEL
LIN {X 0,Y 453.466,Z 417.003,A -85,B 0,C 180,E1 -8401.8,E2 -8401.8} C_VEL
LIN {X 0,Y 453.481,Z 416.999,A -85,B 0,C 180,E1 -8404.989,E2 -8404.989} C_VEL
LIN {X 0,Y 453.461,Z 416.999,A -85,B 0,C 180,E1 -8408.312,E2 -8408.312} C_VEL
LIN {X 0,Y 453.495,Z 416.995,A -85,B 0,C 180,E1 -8410.609,E2 -8410.609} C_VEL
LIN {X 0,Y 453.465,Z 416.998,A -85,B 0,C 180,E1 -8414.221,E2 -8414.221} C_VEL
LIN {X 0,Y 453.466,Z 417,A -85,B 0,C 180,E1 -8417.005,E2 -8417.005} C_VEL
LIN {X 0,Y 453.508,Z 416.994,A -85,B 0,C 180,E1 -8420.552,E2 -8420.552} C_VEL
LIN {X 0,Y 453.457,Z 416.998,A -85,B 0,C 180,E1 -8423.917,E2 -8423.917} C_VEL
LIN {X 0,Y 453.485,Z 416.998,A -85,B 0,C 180,E1 -8427.151,E2 -8427.151} C_VEL
LIN {X 0,Y 453.477,Z 416.998,A -85,B 0,C 180,E1 -8430.268,E2 -8430.268} C_VEL
LIN {X 0,Y 453.504,Z 416.997,A -85,B 0,C 180,E1 -8433.294,E2 -8433.294} C_VEL
LIN {X 0,Y 453.5,Z 416.999,A -85,B 0,C 180,E1 -8436.239,E2 -8436.239} C_VEL
LIN {X 0,Y 453.485,Z 416.999,A -85,B 0,C 180,E1 -8439.118,E2 -8439.118} C_VEL
LIN {X 0,Y 453.529,Z 416.995,A -85,B 0,C 180,E1 -8442.365,E2 -8442.365} C_VEL
LIN {X 0,Y 455.628,Z 422.555,A -85,B 0,C 180,E1 -8442.599,E2 -8442.599} C_VEL
LIN {X 0,Y 458.168,Z 429.143,A -85,B 0,C 180,E1 -8442.862,E2 -8442.862} C_VEL
LIN {X 0,Y 456.906,Z 505.141,A -85,B 0,C 180,E1 -8444.327,E2 -8444.327} C_VEL
LIN {X 0,Y 456.759,Z 522.399,A -85,B 0,C 180,E1 -8444.694,E2 -8444.694} C_VEL
LIN {X 0,Y 456.471,Z 534.517,A -85,B 0,C 180,E1 -8445.112,E2 -8445.112} C_VEL
LIN {X 0,Y 456.186,Z 546.955,A -85,B 0,C 180,E1 -8445.73,E2 -8445.73} C_VEL
LIN {X 0,Y 455.75,Z 558.713,A -85,B 0,C 180,E1 -8446.496,E2 -8446.496} C_VEL
LIN {X 0,Y 455.318,Z 569.644,A -85,B 0,C 180,E1 -8447.407,E2 -8447.407} C_VEL
LIN {X 0,Y 454.882,Z 579.335,A -85,B 0,C 180,E1 -8448.413,E2 -8448.413} C_VEL
LIN {X 0,Y 454.44,Z 588.135,A -85,B 0,C 180,E1 -8449.53,E2 -8449.53} C_VEL
LIN {X 0,Y 453.966,Z 596.689,A -85,B 0,C 180,E1 -8450.869,E2 -8450.869} C_VEL
LIN {X 0,Y 453.602,Z 603.569,A -85,B 0,C 180,E1 -8452.231,E2 -8452.231} C_VEL
LIN {X 0,Y 453.194,Z 609.684,A -85,B 0,C 180,E1 -8453.768,E2 -8453.768} C_VEL
LIN {X 0,Y 453.149,Z 613.676,A -85,B 0,C 180,E1 -8455.107,E2 -8455.107} C_VEL
LIN {X 0,Y 452.956,Z 616.608,A -85,B 0,C 180,E1 -8456.442,E2 -8456.442} C_VEL
LIN {X 0,Y 452.768,Z 618.016,A -85,B 0,C 180,E1 -8457.331,E2 -8457.331} C_VEL
LIN {X 0,Y 452.669,Z 618.977,A -85,B 0,C 180,E1 -8458.221,E2 -8458.221} C_VEL
LIN {X 0,Y 452.628,Z 619.536,A -85,B 0,C 180,E1 -8459.11,E2 -8459.11} C_VEL
LIN {X 0,Y 452.613,Z 619.695,A -85,B 0,C 180,E1 -8460,E2 -8460} C_VEL
LIN {X 0,Y 452.612,Z 619.407,A -85,B 0,C 180,E1 -8460.89,E2 -8460.89} C_VEL
LIN {X 0,Y 452.641,Z 618.716,A -85,B 0,C 180,E1 -8461.78,E2 -8461.78} C_VEL
LIN {X 0,Y 452.756,Z 617.617,A -85,B 0,C 180,E1 -8462.669,E2 -8462.669} C_VEL
LIN {X 0,Y 452.946,Z 616.09,A -85,B 0,C 180,E1 -8463.558,E2 -8463.558} C_VEL
LIN {X 0,Y 453.019,Z 612.98,A -85,B 0,C 180,E1 -8464.895,E2 -8464.895} C_VEL
LIN {X 0,Y 453.083,Z 608.793,A -85,B 0,C 180,E1 -8466.234,E2 -8466.234} C_VEL
LIN {X 0,Y 453.371,Z 602.364,A -85,B 0,C 180,E1 -8467.796,E2 -8467.796} C_VEL
LIN {X 0,Y 453.734,Z 595.354,A -85,B 0,C 180,E1 -8469.135,E2 -8469.135} C_VEL
LIN {X 0,Y 454.052,Z 588.192,A -85,B 0,C 180,E1 -8470.253,E2 -8470.253} C_VEL
LIN {X 0,Y 454.485,Z 579.519,A -85,B 0,C 180,E1 -8471.371,E2 -8471.371} C_VEL
LIN {X 0,Y 454.932,Z 568.805,A -85,B 0,C 180,E1 -8472.491,E2 -8472.491} C_VEL
LIN {X 0,Y 455.393,Z 558.171,A -85,B 0,C 180,E1 -8473.385,E2 -8473.385} C_VEL
LIN {X 0,Y 455.762,Z 546.385,A -85,B 0,C 180,E1 -8474.17,E2 -8474.17} C_VEL
LIN {X 0,Y 456.086,Z 534.2,A -85,B 0,C 180,E1 -8474.787,E2 -8474.787} C_VEL
LIN {X 0,Y 456.429,Z 521.078,A -85,B 0,C 180,E1 -8475.26,E2 -8475.26} C_VEL
LIN {X 0,Y 456.542,Z 506.989,A -85,B 0,C 180,E1 -8475.571,E2 -8475.571} C_VEL
LIN {X 0,Y 457.404,Z 428.44,A -85,B 0,C 180,E1 -8476.969,E2 -8476.969} C_VEL
LIN {X 0,Y 453.518,Z 416.997,A -85,B 0,C 180,E1 -8477.327,E2 -8477.327} C_VEL
LIN {X 0,Y 453.505,Z 416.997,A -85,B 0,C 180,E1 -8479.934,E2 -8479.934} C_VEL
LIN {X 0,Y 453.481,Z 416.994,A -85,B 0,C 180,E1 -8482.796,E2 -8482.796} C_VEL
LIN {X 0,Y 453.499,Z 416.992,A -85,B 0,C 180,E1 -8485.993,E2 -8485.993} C_VEL
LIN {X 0,Y 453.511,Z 416.989,A -85,B 0,C 180,E1 -8488.712,E2 -8488.712} C_VEL
LIN {X 0,Y 453.467,Z 416.991,A -85,B 0,C 180,E1 -8491.799,E2 -8491.799} C_VEL
LIN {X 0,Y 453.483,Z 416.989,A -85,B 0,C 180,E1 -8494.989,E2 -8494.989} C_VEL
LIN {X 0,Y 453.466,Z 416.998,A -85,B 0,C 180,E1 -8498.312,E2 -8498.312} C_VEL
LIN {X 0,Y 453.496,Z 416.987,A -85,B 0,C 180,E1 -8500.609,E2 -8500.609} C_VEL
LIN {X 0,Y 453.459,Z 417.002,A -85,B 0,C 180,E1 -8503.244,E2 -8503.244} C_VEL
LIN {X 0,Y 453.469,Z 416.988,A -85,B 0,C 180,E1 -8505.779,E2 -8505.779} C_VEL
LIN {X 0,Y 453.482,Z 416.997,A -85,B 0,C 180,E1 -8508.209,E2 -8508.209} C_VEL
LIN {X 0,Y 453.493,Z 416.996,A -85,B 0,C 180,E1 -8510.794,E2 -8510.794} C_VEL
LIN {X 0,Y 453.454,Z 416.997,A -85,B 0,C 180,E1 -8513.917,E2 -8513.917} C_VEL
LIN {X 0,Y 453.486,Z 416.996,A -85,B 0,C 180,E1 -8517.151,E2 -8517.151} C_VEL
LIN {X 0,Y 453.465,Z 417.004,A -85,B 0,C 180,E1 -8520.267,E2 -8520.267} C_VEL
LIN {X 0,Y 453.472,Z 417.046,A -85,B 0,C 180,E1 -8523.523,E2 -8523.523} C_VEL
LIN {X 0,Y 455.893,Z 428.741,A -85,B 0,C 180,E1 -8525.637,E2 -8525.637} C_VEL
LIN {X 0,Y 456.196,Z 433.098,A -85,B 0,C 180,E1 -8526.387,E2 -8526.387} C_VEL
LIN {X 0,Y 455.999,Z 438.386,A -85,B 0,C 180,E1 -8527.274,E2 -8527.274} C_VEL
LIN {X 0,Y 455.173,Z 442.029,A -85,B 0,C 180,E1 -8527.85,E2 -8527.85} C_VEL
LIN {X 0,Y 449.17,Z 454.506,A -85,B 0,C 180,E1 -8529.657,E2 -8529.657} C_VEL
LIN {X 0,Y 448.381,Z 458.23,A -85,B 0,C 180,E1 -8530.234,E2 -8530.234} C_VEL
LIN {X 0,Y 448.03,Z 470.994,A -85,B 0,C 180,E1 -8532.229,E2 -8532.229} C_VEL
LIN {X 0,Y 450.987,Z 488.811,A -85,B 0,C 180,E1 -8532.648,E2 -8532.648} C_VEL
LIN {X 0,Y 450.077,Z 580.598,A -85,B 0,C 180,E1 -8534.141,E2 -8534.141} C_VEL
LIN {X 0,Y 449.794,Z 594.035,A -85,B 0,C 180,E1 -8534.538,E2 -8534.538} C_VEL
LIN {X 0,Y 449.318,Z 606.582,A -85,B 0,C 180,E1 -8535.101,E2 -8535.101} C_VEL
LIN {X 0,Y 448.805,Z 618.691,A -85,B 0,C 180,E1 -8535.838,E2 -8535.838} C_VEL
LIN {X 0,Y 448.263,Z 630.083,A -85,B 0,C 180,E1 -8536.739,E2 -8536.739} C_VEL
LIN {X 0,Y 447.688,Z 640.402,A -85,B 0,C 180,E1 -8537.765,E2 -8537.765} C_VEL
LIN {X 0,Y 447.063,Z 649.69,A -85,B 0,C 180,E1 -8538.897,E2 -8538.897} C_VEL
LIN {X 0,Y 446.545,Z 658.645,A -85,B 0,C 180,E1 -8540.259,E2 -8540.259} C_VEL
LIN {X 0,Y 446.105,Z 665.833,A -85,B 0,C 180,E1 -8541.621,E2 -8541.621} C_VEL
LIN {X 0,Y 445.8,Z 671.819,A -85,B 0,C 180,E1 -8543.041,E2 -8543.041} C_VEL
LIN {X 0,Y 445.649,Z 676.761,A -85,B 0,C 180,E1 -8544.57,E2 -8544.57} C_VEL
LIN {X 0,Y 445.49,Z 679.043,A -85,B 0,C 180,E1 -8545.476,E2 -8545.476} C_VEL
LIN {X 0,Y 445.504,Z 680.9,A -85,B 0,C 180,E1 -8546.382,E2 -8546.382} C_VEL
LIN {X 0,Y 445.462,Z 682.324,A -85,B 0,C 180,E1 -8547.287,E2 -8547.287} C_VEL
LIN {X 0,Y 445.341,Z 683.937,A -85,B 0,C 180,E1 -8549.096,E2 -8549.096} C_VEL
LIN {X 0,Y 445.342,Z 684.174,A -85,B 0,C 180,E1 -8550,E2 -8550} C_VEL
LIN {X 0,Y 445.341,Z 683.985,A -85,B 0,C 180,E1 -8550.904,E2 -8550.904} C_VEL
LIN {X 0,Y 445.462,Z 682.434,A -85,B 0,C 180,E1 -8552.713,E2 -8552.713} C_VEL
LIN {X 0,Y 445.503,Z 681.072,A -85,B 0,C 180,E1 -8553.618,E2 -8553.618} C_VEL
LIN {X 0,Y 445.536,Z 678.208,A -85,B 0,C 180,E1 -8554.977,E2 -8554.977} C_VEL
LIN {X 0,Y 445.766,Z 674.313,A -85,B 0,C 180,E1 -8556.336,E2 -8556.336} C_VEL
LIN {X 0,Y 445.958,Z 669.27,A -85,B 0,C 180,E1 -8557.698,E2 -8557.698} C_VEL
LIN {X 0,Y 446.305,Z 662.909,A -85,B 0,C 180,E1 -8559.06,E2 -8559.06} C_VEL
LIN {X 0,Y 446.761,Z 655.008,A -85,B 0,C 180,E1 -8560.423,E2 -8560.423} C_VEL
LIN {X 0,Y 447.238,Z 646.936,A -85,B 0,C 180,E1 -8561.558,E2 -8561.558} C_VEL
LIN {X 0,Y 447.909,Z 637.02,A -85,B 0,C 180,E1 -8562.69,E2 -8562.69} C_VEL
LIN {X 0,Y 448.388,Z 626.73,A -85,B 0,C 180,E1 -8563.642,E2 -8563.642} C_VEL
LIN {X 0,Y 448.978,Z 614.984,A -85,B 0,C 180,E1 -8564.504,E2 -8564.504} C_VEL
LIN {X 0,Y 449.486,Z 602.759,A -85,B 0,C 180,E1 -8565.183,E2 -8565.183} C_VEL
LIN {X 0,Y 449.929,Z 589.253,A -85,B 0,C 180,E1 -8565.719,E2 -8565.719} C_VEL
LIN {X 0,Y 450.228,Z 576.79,A -85,B 0,C 180,E1 -8566.028,E2 -8566.028} C_VEL
LIN {X 0,Y 450.949,Z 487.87,A -85,B 0,C 180,E1 -8567.462,E2 -8567.462} C_VEL
LIN {X 0,Y 448.035,Z 470.906,A -85,B 0,C 180,E1 -8567.875,E2 -8567.875} C_VEL
LIN {X 0,Y 448.51,Z 454.975,A -85,B 0,C 180,E1 -8570.405,E2 -8570.405} C_VEL
LIN {X 0,Y 449.177,Z 437.792,A -85,B 0,C 180,E1 -8573.271,E2 -8573.271} C_VEL
LIN {X 0,Y 449.19,Z 431.281,A -85,B 0,C 180,E1 -8574.385,E2 -8574.385} C_VEL
LIN {X 0,Y 446.426,Z 417.88,A -85,B 0,C 180,E1 -8576.837,E2 -8576.837} C_VEL
LIN {X 0,Y 446.431,Z 417.878,A -85,B 0,C 180,E1 -8580.02,E2 -8580.02} C_VEL
LIN {X 0,Y 446.448,Z 417.878,A -85,B 0,C 180,E1 -8583.454,E2 -8583.454} C_VEL
LIN {X 0,Y 446.402,Z 417.88,A -85,B 0,C 180,E1 -8586.745,E2 -8586.745} C_VEL
LIN {X 0,Y 446.445,Z 417.867,A -85,B 0,C 180,E1 -8590.198,E2 -8590.198} C_VEL
LIN {X 0,Y 446.432,Z 417.875,A -85,B 0,C 180,E1 -8592.605,E2 -8592.605} C_VEL
LIN {X 0,Y 446.458,Z 417.875,A -85,B 0,C 180,E1 -8595.103,E2 -8595.103} C_VEL
LIN {X 0,Y 446.431,Z 417.87,A -85,B 0,C 180,E1 -8598.609,E2 -8598.609} C_VEL
LIN {X 0,Y 446.458,Z 417.875,A -85,B 0,C 180,E1 -8600.974,E2 -8600.974} C_VEL
LIN {X 0,Y 446.42,Z 417.868,A -85,B 0,C 180,E1 -8604.374,E2 -8604.374} C_VEL
LIN {X 0,Y 446.425,Z 417.874,A -85,B 0,C 180,E1 -8607.638,E2 -8607.638} C_VEL
LIN {X 0,Y 446.426,Z 417.878,A -85,B 0,C 180,E1 -8610.789,E2 -8610.789} C_VEL
LIN {X 0,Y 446.459,Z 418.042,A -85,B 0,C 180,E1 -8613.401,E2 -8613.401} C_VEL
LIN {X 0,Y 449.026,Z 430.769,A -85,B 0,C 180,E1 -8615.657,E2 -8615.657} C_VEL
LIN {X 0,Y 449.292,Z 435.69,A -85,B 0,C 180,E1 -8616.492,E2 -8616.492} C_VEL
LIN {X 0,Y 448.494,Z 457.528,A -85,B 0,C 180,E1 -8620.088,E2 -8620.088} C_VEL
LIN {X 0,Y 447.941,Z 471.441,A -85,B 0,C 180,E1 -8622.363,E2 -8622.363} C_VEL
LIN {X 0,Y 450.585,Z 488.118,A -85,B 0,C 180,E1 -8622.783,E2 -8622.783} C_VEL
LIN {X 0,Y 449.426,Z 581.556,A -85,B 0,C 180,E1 -8624.496,E2 -8624.496} C_VEL
LIN {X 0,Y 449.001,Z 595.442,A -85,B 0,C 180,E1 -8624.946,E2 -8624.946} C_VEL
LIN {X 0,Y 448.615,Z 608.002,A -85,B 0,C 180,E1 -8625.541,E2 -8625.541} C_VEL
LIN {X 0,Y 448.111,Z 619.667,A -85,B 0,C 180,E1 -8626.278,E2 -8626.278} C_VEL
LIN {X 0,Y 447.739,Z 630.628,A -85,B 0,C 180,E1 -8627.155,E2 -8627.155} C_VEL
LIN {X 0,Y 447.172,Z 641.172,A -85,B 0,C 180,E1 -8628.21,E2 -8628.21} C_VEL
LIN {X 0,Y 446.72,Z 650.416,A -85,B 0,C 180,E1 -8629.347,E2 -8629.347} C_VEL
LIN {X 0,Y 446.321,Z 658.025,A -85,B 0,C 180,E1 -8630.483,E2 -8630.483} C_VEL
LIN {X 0,Y 445.972,Z 665.438,A -85,B 0,C 180,E1 -8631.846,E2 -8631.846} C_VEL
LIN {X 0,Y 445.709,Z 672.18,A -85,B 0,C 180,E1 -8633.412,E2 -8633.412} C_VEL
LIN {X 0,Y 445.61,Z 676.057,A -85,B 0,C 180,E1 -8634.57,E2 -8634.57} C_VEL
LIN {X 0,Y 445.478,Z 678.536,A -85,B 0,C 180,E1 -8635.476,E2 -8635.476} C_VEL
LIN {X 0,Y 445.481,Z 680.521,A -85,B 0,C 180,E1 -8636.382,E2 -8636.382} C_VEL
LIN {X 0,Y 445.461,Z 682.09,A -85,B 0,C 180,E1 -8637.287,E2 -8637.287} C_VEL
LIN {X 0,Y 445.379,Z 683.203,A -85,B 0,C 180,E1 -8638.191,E2 -8638.191} C_VEL
LIN {X 0,Y 445.341,Z 683.889,A -85,B 0,C 180,E1 -8639.096,E2 -8639.096} C_VEL
LIN {X 0,Y 445.342,Z 684.18,A -85,B 0,C 180,E1 -8640,E2 -8640} C_VEL
LIN {X 0,Y 445.341,Z 684.031,A -85,B 0,C 180,E1 -8640.904,E2 -8640.904} C_VEL
LIN {X 0,Y 445.379,Z 683.453,A -85,B 0,C 180,E1 -8641.808,E2 -8641.808} C_VEL
LIN {X 0,Y 445.461,Z 682.477,A -85,B 0,C 180,E1 -8642.713,E2 -8642.713} C_VEL
LIN {X 0,Y 445.5,Z 681.056,A -85,B 0,C 180,E1 -8643.618,E2 -8643.618} C_VEL
LIN {X 0,Y 445.53,Z 678.083,A -85,B 0,C 180,E1 -8644.977,E2 -8644.977} C_VEL
LIN {X 0,Y 445.726,Z 674.019,A -85,B 0,C 180,E1 -8646.337,E2 -8646.337} C_VEL
LIN {X 0,Y 445.959,Z 667.78,A -85,B 0,C 180,E1 -8647.926,E2 -8647.926} C_VEL
LIN {X 0,Y 446.329,Z 660.882,A -85,B 0,C 180,E1 -8649.288,E2 -8649.288} C_VEL
LIN {X 0,Y 446.79,Z 652.278,A -85,B 0,C 180,E1 -8650.651,E2 -8650.651} C_VEL
LIN {X 0,Y 447.233,Z 643.423,A -85,B 0,C 180,E1 -8651.788,E2 -8651.788} C_VEL
LIN {X 0,Y 447.857,Z 631.804,A -85,B 0,C 180,E1 -8652.985,E2 -8652.985} C_VEL
LIN {X 0,Y 448.291,Z 621.516,A -85,B 0,C 180,E1 -8653.832,E2 -8653.832} C_VEL
LIN {X 0,Y 448.844,Z 608.279,A -85,B 0,C 180,E1 -8654.683,E2 -8654.683} C_VEL
LIN {X 0,Y 449.307,Z 595.694,A -85,B 0,C 180,E1 -8655.276,E2 -8655.276} C_VEL
LIN {X 0,Y 449.674,Z 582.864,A -85,B 0,C 180,E1 -8655.699,E2 -8655.699} C_VEL
LIN {X 0,Y 451.149,Z 487.594,A -85,B 0,C 180,E1 -8657.57,E2 -8657.57} C_VEL
LIN {X 0,Y 448.495,Z 472.514,A -85,B 0,C 180,E1 -8658.033,E2 -8658.033} C_VEL
LIN {X 0,Y 449.147,Z 453.562,A -85,B 0,C 180,E1 -8661.094,E2 -8661.094} C_VEL
LIN {X 0,Y 449.792,Z 434.275,A -85,B 0,C 180,E1 -8664.173,E2 -8664.173} C_VEL
LIN {X 0,Y 448.202,Z 425.007,A -85,B 0,C 180,E1 -8665.794,E2 -8665.794} C_VEL
LIN {X 0,Y 446.431,Z 417.878,A -85,B 0,C 180,E1 -8667.079,E2 -8667.079} C_VEL
LIN {X 0,Y 446.427,Z 417.88,A -85,B 0,C 180,E1 -8670.25,E2 -8670.25} C_VEL
LIN {X 0,Y 446.447,Z 417.876,A -85,B 0,C 180,E1 -8673.454,E2 -8673.454} C_VEL
LIN {X 0,Y 446.402,Z 417.878,A -85,B 0,C 180,E1 -8676.745,E2 -8676.745} C_VEL
LIN {X 0,Y 446.457,Z 417.872,A -85,B 0,C 180,E1 -8679.525,E2 -8679.525} C_VEL
LIN {X 0,Y 446.432,Z 417.876,A -85,B 0,C 180,E1 -8682.605,E2 -8682.605} C_VEL
LIN {X 0,Y 446.456,Z 417.873,A -85,B 0,C 180,E1 -8685.103,E2 -8685.103} C_VEL
LIN {X 0,Y 446.43,Z 417.876,A -85,B 0,C 180,E1 -8688.609,E2 -8688.609} C_VEL
LIN {X 0,Y 446.446,Z 417.873,A -85,B 0,C 180,E1 -8690.973,E2 -8690.973} C_VEL
LIN {X 0,Y 446.419,Z 417.876,A -85,B 0,C 180,E1 -8694.374,E2 -8694.374} C_VEL
LIN {X 0,Y 446.424,Z 417.875,A -85,B 0,C 180,E1 -8697.638,E2 -8697.638} C_VEL
LIN {X 0,Y 446.455,Z 417.958,A -85,B 0,C 180,E1 -8700.572,E2 -8700.572} C_VEL
LIN {X 0,Y 449.916,Z 434.222,A -85,B 0,C 180,E1 -8703.381,E2 -8703.381} C_VEL
LIN {X 0,Y 449.665,Z 444.682,A -85,B 0,C 180,E1 -8705.039,E2 -8705.039} C_VEL
LIN {X 0,Y 448.529,Z 466.313,A -85,B 0,C 180,E1 -8708.394,E2 -8708.394} C_VEL
LIN {X 0,Y 447.503,Z 489.483,A -85,B 0,C 180,E1 -8711.954,E2 -8711.954} C_VEL
LIN {X 0,Y 447.436,Z 491.339,A -85,B 0,C 180,E1 -8712.238,E2 -8712.238} C_VEL
LIN {X 0,Y 450.42,Z 516.413,A -85,B 0,C 180,E1 -8712.828,E2 -8712.828} C_VEL
LIN {X 0,Y 449.986,Z 555.72,A -85,B 0,C 180,E1 -8713.512,E2 -8713.512} C_VEL
LIN {X 0,Y 449.419,Z 605.535,A -85,B 0,C 180,E1 -8714.321,E2 -8714.321} C_VEL
LIN {X 0,Y 449.137,Z 618.679,A -85,B 0,C 180,E1 -8714.718,E2 -8714.718} C_VEL
LIN {X 0,Y 448.653,Z 630.734,A -85,B 0,C 180,E1 -8715.253,E2 -8715.253} C_VEL
LIN {X 0,Y 448.159,Z 642.089,A -85,B 0,C 180,E1 -8715.932,E2 -8715.932} C_VEL
LIN {X 0,Y 447.619,Z 653.681,A -85,B 0,C 180,E1 -8716.837,E2 -8716.837} C_VEL
LIN {X 0,Y 447.058,Z 664.159,A -85,B 0,C 180,E1 -8717.862,E2 -8717.862} C_VEL
LIN {X 0,Y 446.616,Z 672.674,A -85,B 0,C 180,E1 -8718.886,E2 -8718.886} C_VEL
LIN {X 0,Y 446.22,Z 680.497,A -85,B 0,C 180,E1 -8720.023,E2 -8720.023} C_VEL
LIN {X 0,Y 445.882,Z 688.111,A -85,B 0,C 180,E1 -8721.388,E2 -8721.388} C_VEL
LIN {X 0,Y 445.636,Z 694.22,A -85,B 0,C 180,E1 -8722.752,E2 -8722.752} C_VEL
LIN {X 0,Y 445.5,Z 699.41,A -85,B 0,C 180,E1 -8724.231,E2 -8724.231} C_VEL
LIN {X 0,Y 445.469,Z 702.725,A -85,B 0,C 180,E1 -8725.476,E2 -8725.476} C_VEL
LIN {X 0,Y 445.485,Z 704.622,A -85,B 0,C 180,E1 -8726.382,E2 -8726.382} C_VEL
LIN {X 0,Y 445.489,Z 706.055,A -85,B 0,C 180,E1 -8727.287,E2 -8727.287} C_VEL
LIN {X 0,Y 445.405,Z 707.679,A -85,B 0,C 180,E1 -8729.096,E2 -8729.096} C_VEL
LIN {X 0,Y 445.419,Z 707.901,A -85,B 0,C 180,E1 -8730,E2 -8730} C_VEL
LIN {X 0,Y 445.405,Z 707.679,A -85,B 0,C 180,E1 -8730.904,E2 -8730.904} C_VEL
LIN {X 0,Y 445.492,Z 706.054,A -85,B 0,C 180,E1 -8732.713,E2 -8732.713} C_VEL
LIN {X 0,Y 445.495,Z 704.621,A -85,B 0,C 180,E1 -8733.618,E2 -8733.618} C_VEL
LIN {X 0,Y 445.513,Z 701.638,A -85,B 0,C 180,E1 -8734.977,E2 -8734.977} C_VEL
LIN {X 0,Y 445.577,Z 697.227,A -85,B 0,C 180,E1 -8736.44,E2 -8736.44} C_VEL
LIN {X 0,Y 445.748,Z 691.334,A -85,B 0,C 180,E1 -8737.93,E2 -8737.93} C_VEL
LIN {X 0,Y 446.051,Z 684.51,A -85,B 0,C 180,E1 -8739.294,E2 -8739.294} C_VEL
LIN {X 0,Y 446.349,Z 677.522,A -85,B 0,C 180,E1 -8740.432,E2 -8740.432} C_VEL
LIN {X 0,Y 446.834,Z 669.076,A -85,B 0,C 180,E1 -8741.568,E2 -8741.568} C_VEL
LIN {X 0,Y 447.362,Z 658.609,A -85,B 0,C 180,E1 -8742.705,E2 -8742.705} C_VEL
LIN {X 0,Y 447.852,Z 648.226,A -85,B 0,C 180,E1 -8743.615,E2 -8743.615} C_VEL
LIN {X 0,Y 448.418,Z 636.761,A -85,B 0,C 180,E1 -8744.407,E2 -8744.407} C_VEL
LIN {X 0,Y 448.913,Z 624.825,A -85,B 0,C 180,E1 -8745.028,E2 -8745.028} C_VEL
LIN {X 0,Y 449.353,Z 611.883,A -85,B 0,C 180,E1 -8745.507,E2 -8745.507} C_VEL
LIN {X 0,Y 449.596,Z 599.558,A -85,B 0,C 180,E1 -8745.789,E2 -8745.789} C_VEL
LIN {X 0,Y 449.999,Z 562.251,A -85,B 0,C 180,E1 -8746.42,E2 -8746.42} C_VEL
LIN {X 0,Y 450.683,Z 515.236,A -85,B 0,C 180,E1 -8747.34,E2 -8747.34} C_VEL
LIN {X 0,Y 447.649,Z 489.253,A -85,B 0,C 180,E1 -8748.032,E2 -8748.032} C_VEL
LIN {X 0,Y 447.312,Z 486.913,A -85,B 0,C 180,E1 -8748.103,E2 -8748.103} C_VEL
LIN {X 0,Y 448.255,Z 465.911,A -85,B 0,C 180,E1 -8751.379,E2 -8751.379} C_VEL
LIN {X 0,Y 449.445,Z 443.526,A -85,B 0,C 180,E1 -8754.974,E2 -8754.974} C_VEL
LIN {X 0,Y 449.973,Z 434.734,A -85,B 0,C 180,E1 -8756.432,E2 -8756.432} C_VEL
LIN {X 0,Y 448.127,Z 424.782,A -85,B 0,C 180,E1 -8758.294,E2 -8758.294} C_VEL
LIN {X 0,Y 446.431,Z 417.882,A -85,B 0,C 180,E1 -8759.712,E2 -8759.712} C_VEL
LIN {X 0,Y 446.424,Z 417.878,A -85,B 0,C 180,E1 -8762.362,E2 -8762.362} C_VEL
LIN {X 0,Y 446.419,Z 417.881,A -85,B 0,C 180,E1 -8765.626,E2 -8765.626} C_VEL
LIN {X 0,Y 446.438,Z 417.876,A -85,B 0,C 180,E1 -8769.028,E2 -8769.028} C_VEL
LIN {X 0,Y 446.423,Z 417.874,A -85,B 0,C 180,E1 -8772.275,E2 -8772.275} C_VEL
LIN {X 0,Y 446.455,Z 417.874,A -85,B 0,C 180,E1 -8775.104,E2 -8775.104} C_VEL
LIN {X 0,Y 446.43,Z 417.874,A -85,B 0,C 180,E1 -8778.609,E2 -8778.609} C_VEL
LIN {X 0,Y 446.458,Z 417.874,A -85,B 0,C 180,E1 -8780.974,E2 -8780.974} C_VEL
LIN {X 0,Y 446.422,Z 417.875,A -85,B 0,C 180,E1 -8784.374,E2 -8784.374} C_VEL
LIN {X 0,Y 446.425,Z 417.876,A -85,B 0,C 180,E1 -8787.639,E2 -8787.639} C_VEL
LIN {X 0,Y 446.451,Z 417.876,A -85,B 0,C 180,E1 -8790.791,E2 -8790.791} C_VEL
LIN {X 0,Y 446.48,Z 417.87,A -85,B 0,C 180,E1 -8793.849,E2 -8793.849} C_VEL
LIN {X 0,Y 446.429,Z 417.88,A -85,B 0,C 180,E1 -8796.823,E2 -8796.823} C_VEL
LIN {X 0,Y 446.446,Z 417.875,A -85,B 0,C 180,E1 -8799.737,E2 -8799.737} C_VEL
LIN {X 0,Y 446.474,Z 417.874,A -85,B 0,C 180,E1 -8802.002,E2 -8802.002} C_VEL
LIN {X 0,Y 448.04,Z 422.108,A -85,B 0,C 180,E1 -8802.192,E2 -8802.192} C_VEL
LIN {X 0,Y 451.562,Z 431.241,A -85,B 0,C 180,E1 -8802.582,E2 -8802.582} C_VEL
LIN {X 0,Y 450.019,Z 520.823,A -85,B 0,C 180,E1 -8804.372,E2 -8804.372} C_VEL
LIN {X 0,Y 449.734,Z 533.587,A -85,B 0,C 180,E1 -8804.797,E2 -8804.797} C_VEL
LIN {X 0,Y 449.456,Z 546.012,A -85,B 0,C 180,E1 -8805.396,E2 -8805.396} C_VEL
LIN {X 0,Y 448.986,Z 558.394,A -85,B 0,C 180,E1 -8806.198,E2 -8806.198} C_VEL
LIN {X 0,Y 448.497,Z 569.317,A -85,B 0,C 180,E1 -8807.097,E2 -8807.097} C_VEL
LIN {X 0,Y 448.091,Z 578.248,A -85,B 0,C 180,E1 -8808.006,E2 -8808.006} C_VEL
LIN {X 0,Y 447.591,Z 587.386,A -85,B 0,C 180,E1 -8809.139,E2 -8809.139} C_VEL
LIN {X 0,Y 447.085,Z 596.229,A -85,B 0,C 180,E1 -8810.5,E2 -8810.5} C_VEL
LIN {X 0,Y 446.718,Z 603.298,A -85,B 0,C 180,E1 -8811.86,E2 -8811.86} C_VEL
LIN {X 0,Y 446.365,Z 609.318,A -85,B 0,C 180,E1 -8813.343,E2 -8813.343} C_VEL
LIN {X 0,Y 446.102,Z 613.24,A -85,B 0,C 180,E1 -8814.576,E2 -8814.576} C_VEL
LIN {X 0,Y 446.117,Z 615.5,A -85,B 0,C 180,E1 -8815.482,E2 -8815.482} C_VEL
LIN {X 0,Y 445.921,Z 617.352,A -85,B 0,C 180,E1 -8816.386,E2 -8816.386} C_VEL
LIN {X 0,Y 445.72,Z 618.743,A -85,B 0,C 180,E1 -8817.289,E2 -8817.289} C_VEL
LIN {X 0,Y 445.609,Z 619.693,A -85,B 0,C 180,E1 -8818.192,E2 -8818.192} C_VEL
LIN {X 0,Y 445.565,Z 620.241,A -85,B 0,C 180,E1 -8819.096,E2 -8819.096} C_VEL
LIN {X 0,Y 445.547,Z 620.385,A -85,B 0,C 180,E1 -8820,E2 -8820} C_VEL
LIN {X 0,Y 445.545,Z 620.077,A -85,B 0,C 180,E1 -8820.904,E2 -8820.904} C_VEL
LIN {X 0,Y 445.581,Z 619.363,A -85,B 0,C 180,E1 -8821.808,E2 -8821.808} C_VEL
LIN {X 0,Y 445.708,Z 618.246,A -85,B 0,C 180,E1 -8822.711,E2 -8822.711} C_VEL
LIN {X 0,Y 445.936,Z 615.743,A -85,B 0,C 180,E1 -8824.067,E2 -8824.067} C_VEL
LIN {X 0,Y 446.014,Z 612.241,A -85,B 0,C 180,E1 -8825.425,E2 -8825.425} C_VEL
LIN {X 0,Y 446.189,Z 607.474,A -85,B 0,C 180,E1 -8826.822,E2 -8826.822} C_VEL
LIN {X 0,Y 446.47,Z 600.609,A -85,B 0,C 180,E1 -8828.372,E2 -8828.372} C_VEL
LIN {X 0,Y 446.882,Z 592.975,A -85,B 0,C 180,E1 -8829.733,E2 -8829.733} C_VEL
LIN {X 0,Y 447.263,Z 585.182,A -85,B 0,C 180,E1 -8830.869,E2 -8830.869} C_VEL
LIN {X 0,Y 447.75,Z 575.681,A -85,B 0,C 180,E1 -8832.004,E2 -8832.004} C_VEL
LIN {X 0,Y 448.204,Z 565.297,A -85,B 0,C 180,E1 -8833.01,E2 -8833.01} C_VEL
LIN {X 0,Y 448.619,Z 553.375,A -85,B 0,C 180,E1 -8833.937,E2 -8833.937} C_VEL
LIN {X 0,Y 448.987,Z 540.904,A -85,B 0,C 180,E1 -8834.678,E2 -8834.678} C_VEL
LIN {X 0,Y 449.375,Z 527.168,A -85,B 0,C 180,E1 -8835.274,E2 -8835.274} C_VEL
LIN {X 0,Y 449.581,Z 513.985,A -85,B 0,C 180,E1 -8835.644,E2 -8835.644} C_VEL
LIN {X 0,Y 450.57,Z 429.99,A -85,B 0,C 180,E1 -8837.181,E2 -8837.181} C_VEL
LIN {X 0,Y 446.471,Z 417.876,A -85,B 0,C 180,E1 -8837.58,E2 -8837.58} C_VEL
LIN {X 0,Y 446.446,Z 417.875,A -85,B 0,C 180,E1 -8840.263,E2 -8840.263} C_VEL
LIN {X 0,Y 446.427,Z 417.874,A -85,B 0,C 180,E1 -8843.177,E2 -8843.177} C_VEL
LIN {X 0,Y 446.461,Z 417.868,A -85,B 0,C 180,E1 -8846.198,E2 -8846.198} C_VEL
LIN {X 0,Y 446.45,Z 417.875,A -85,B 0,C 180,E1 -8849.209,E2 -8849.209} C_VEL
LIN {X 0,Y 446.425,Z 417.868,A -85,B 0,C 180,E1 -8852.362,E2 -8852.362} C_VEL
LIN {X 0,Y 446.422,Z 417.875,A -85,B 0,C 180,E1 -8855.626,E2 -8855.626} C_VEL
LIN {X 0,Y 446.444,Z 417.871,A -85,B 0,C 180,E1 -8859.027,E2 -8859.027} C_VEL
LIN {X 0,Y 446.437,Z 417.872,A -85,B 0,C 180,E1 -8862.277,E2 -8862.277} C_VEL
LIN {X 0,Y 446.456,Z 417.865,A -85,B 0,C 180,E1 -8865.103,E2 -8865.103} C_VEL
LIN {X 0,Y 446.431,Z 417.878,A -85,B 0,C 180,E1 -8868.609,E2 -8868.609} C_VEL
LIN {X 0,Y 446.444,Z 417.876,A -85,B 0,C 180,E1 -8870.973,E2 -8870.973} C_VEL
LIN {X 0,Y 446.42,Z 417.878,A -85,B 0,C 180,E1 -8874.374,E2 -8874.374} C_VEL
LIN {X 0,Y 446.425,Z 417.875,A -85,B 0,C 180,E1 -8877.638,E2 -8877.638} C_VEL
LIN {X 0,Y 446.424,Z 417.882,A -85,B 0,C 180,E1 -8880.789,E2 -8880.789} C_VEL
LIN {X 0,Y 446.421,Z 417.984,A -85,B 0,C 180,E1 -8883.295,E2 -8883.295} C_VEL
LIN {X 0,Y 449.063,Z 430.645,A -85,B 0,C 180,E1 -8885.616,E2 -8885.616} C_VEL
LIN {X 0,Y 449.216,Z 435.729,A -85,B 0,C 180,E1 -8886.487,E2 -8886.487} C_VEL
LIN {X 0,Y 448.496,Z 455.765,A -85,B 0,C 180,E1 -8889.834,E2 -8889.834} C_VEL
LIN {X 0,Y 448.381,Z 458.23,A -85,B 0,C 180,E1 -8890.234,E2 -8890.234} C_VEL
LIN {X 0,Y 447.576,Z 461.213,A -85,B 0,C 180,E1 -8890.664,E2 -8890.664} C_VEL
LIN {X 0,Y 444.4,Z 466.094,A -85,B 0,C 180,E1 -8891.313,E2 -8891.313} C_VEL
LIN {X 0,Y 441.669,Z 470.608,A -85,B 0,C 180,E1 -8891.85,E2 -8891.85} C_VEL
LIN {X 0,Y 441.474,Z 473.037,A -85,B 0,C 180,E1 -8891.994,E2 -8891.994} C_VEL
LIN {X 0,Y 444.197,Z 488.906,A -85,B 0,C 180,E1 -8892.375,E2 -8892.375} C_VEL
LIN {X 0,Y 443.31,Z 579.431,A -85,B 0,C 180,E1 -8893.863,E2 -8893.863} C_VEL
LIN {X 0,Y 443.016,Z 592.56,A -85,B 0,C 180,E1 -8894.236,E2 -8894.236} C_VEL
LIN {X 0,Y 442.587,Z 604.604,A -85,B 0,C 180,E1 -8894.752,E2 -8894.752} C_VEL
LIN {X 0,Y 442.063,Z 615.496,A -85,B 0,C 180,E1 -8895.381,E2 -8895.381} C_VEL
LIN {X 0,Y 441.48,Z 627.59,A -85,B 0,C 180,E1 -8896.293,E2 -8896.293} C_VEL
LIN {X 0,Y 440.893,Z 638.518,A -85,B 0,C 180,E1 -8897.339,E2 -8897.339} C_VEL
LIN {X 0,Y 440.202,Z 648.146,A -85,B 0,C 180,E1 -8898.488,E2 -8898.488} C_VEL
LIN {X 0,Y 439.623,Z 657.5,A -85,B 0,C 180,E1 -8899.872,E2 -8899.872} C_VEL
LIN {X 0,Y 439.164,Z 664.933,A -85,B 0,C 180,E1 -8901.255,E2 -8901.255} C_VEL
LIN {X 0,Y 438.788,Z 670.9,A -85,B 0,C 180,E1 -8902.638,E2 -8902.638} C_VEL
LIN {X 0,Y 438.68,Z 675.616,A -85,B 0,C 180,E1 -8904.023,E2 -8904.023} C_VEL
LIN {X 0,Y 438.414,Z 679.232,A -85,B 0,C 180,E1 -8905.403,E2 -8905.403} C_VEL
LIN {X 0,Y 438.407,Z 681.09,A -85,B 0,C 180,E1 -8906.323,E2 -8906.323} C_VEL
LIN {X 0,Y 438.392,Z 682.512,A -85,B 0,C 180,E1 -8907.243,E2 -8907.243} C_VEL
LIN {X 0,Y 438.255,Z 684.126,A -85,B 0,C 180,E1 -8909.081,E2 -8909.081} C_VEL
LIN {X 0,Y 438.254,Z 684.363,A -85,B 0,C 180,E1 -8910,E2 -8910} C_VEL
LIN {X 0,Y 438.255,Z 684.173,A -85,B 0,C 180,E1 -8910.919,E2 -8910.919} C_VEL
LIN {X 0,Y 438.392,Z 682.621,A -85,B 0,C 180,E1 -8912.757,E2 -8912.757} C_VEL
LIN {X 0,Y 438.406,Z 681.26,A -85,B 0,C 180,E1 -8913.677,E2 -8913.677} C_VEL
LIN {X 0,Y 438.478,Z 678.395,A -85,B 0,C 180,E1 -8915.057,E2 -8915.057} C_VEL
LIN {X 0,Y 438.687,Z 673.799,A -85,B 0,C 180,E1 -8916.647,E2 -8916.647} C_VEL
LIN {X 0,Y 439.01,Z 667.489,A -85,B 0,C 180,E1 -8918.284,E2 -8918.284} C_VEL
LIN {X 0,Y 439.431,Z 660.668,A -85,B 0,C 180,E1 -8919.668,E2 -8919.668} C_VEL
LIN {X 0,Y 439.953,Z 652.133,A -85,B 0,C 180,E1 -8921.052,E2 -8921.052} C_VEL
LIN {X 0,Y 440.563,Z 643.391,A -85,B 0,C 180,E1 -8922.203,E2 -8922.203} C_VEL
LIN {X 0,Y 441.186,Z 633.641,A -85,B 0,C 180,E1 -8923.252,E2 -8923.252} C_VEL
LIN {X 0,Y 441.679,Z 623.179,A -85,B 0,C 180,E1 -8924.161,E2 -8924.161} C_VEL
LIN {X 0,Y 442.251,Z 611.417,A -85,B 0,C 180,E1 -8924.965,E2 -8924.965} C_VEL
LIN {X 0,Y 442.827,Z 599.229,A -85,B 0,C 180,E1 -8925.594,E2 -8925.594} C_VEL
LIN {X 0,Y 443.139,Z 586.481,A -85,B 0,C 180,E1 -8926.055,E2 -8926.055} C_VEL
LIN {X 0,Y 443.459,Z 573.505,A -85,B 0,C 180,E1 -8926.338,E2 -8926.338} C_VEL
LIN {X 0,Y 444.061,Z 487.922,A -85,B 0,C 180,E1 -8927.741,E2 -8927.741} C_VEL
LIN {X 0,Y 441.142,Z 471.141,A -85,B 0,C 180,E1 -8928.147,E2 -8928.147} C_VEL
LIN {X 0,Y 441.635,Z 454.926,A -85,B 0,C 180,E1 -8930.737,E2 -8930.737} C_VEL
LIN {X 0,Y 442.339,Z 437.614,A -85,B 0,C 180,E1 -8933.652,E2 -8933.652} C_VEL
LIN {X 0,Y 442.358,Z 433.281,A -85,B 0,C 180,E1 -8934.398,E2 -8934.398} C_VEL
LIN {X 0,Y 439.637,Z 419.925,A -85,B 0,C 180,E1 -8936.847,E2 -8936.847} C_VEL
LIN {X 0,Y 439.404,Z 418.756,A -85,B 0,C 180,E1 -8937.087,E2 -8937.087} C_VEL
LIN {X 0,Y 439.381,Z 418.755,A -85,B 0,C 180,E1 -8940.26,E2 -8940.26} C_VEL
LIN {X 0,Y 439.399,Z 418.757,A -85,B 0,C 180,E1 -8943.724,E2 -8943.724} C_VEL
LIN {X 0,Y 439.349,Z 418.76,A -85,B 0,C 180,E1 -8946.887,E2 -8946.887} C_VEL
LIN {X 0,Y 439.404,Z 418.746,A -85,B 0,C 180,E1 -8949.849,E2 -8949.849} C_VEL
LIN {X 0,Y 439.385,Z 418.754,A -85,B 0,C 180,E1 -8952.627,E2 -8952.627} C_VEL
LIN {X 0,Y 439.408,Z 418.754,A -85,B 0,C 180,E1 -8955.271,E2 -8955.271} C_VEL
LIN {X 0,Y 439.391,Z 418.748,A -85,B 0,C 180,E1 -8958.743,E2 -8958.743} C_VEL
LIN {X 0,Y 439.378,Z 418.751,A -85,B 0,C 180,E1 -8961.607,E2 -8961.607} C_VEL
LIN {X 0,Y 439.401,Z 418.749,A -85,B 0,C 180,E1 -8964.844,E2 -8964.844} C_VEL
LIN {X 0,Y 439.375,Z 418.755,A -85,B 0,C 180,E1 -8968.14,E2 -8968.14} C_VEL
LIN {X 0,Y 439.403,Z 418.751,A -85,B 0,C 180,E1 -8971.606,E2 -8971.606} C_VEL
LIN {X 0,Y 439.407,Z 418.808,A -85,B 0,C 180,E1 -8973.17,E2 -8973.17} C_VEL
LIN {X 0,Y 442.125,Z 432.31,A -85,B 0,C 180,E1 -8975.588,E2 -8975.588} C_VEL
LIN {X 0,Y 442.28,Z 438.216,A -85,B 0,C 180,E1 -8976.593,E2 -8976.593} C_VEL
LIN {X 0,Y 441.543,Z 458.182,A -85,B 0,C 180,E1 -8979.901,E2 -8979.901} C_VEL
LIN {X 0,Y 441.028,Z 471.491,A -85,B 0,C 180,E1 -8982.106,E2 -8982.106} C_VEL
LIN {X 0,Y 443.75,Z 489.074,A -85,B 0,C 180,E1 -8982.561,E2 -8982.561} C_VEL
LIN {X 0,Y 442.493,Z 581.823,A -85,B 0,C 180,E1 -8984.306,E2 -8984.306} C_VEL
LIN {X 0,Y 442.072,Z 595.648,A -85,B 0,C 180,E1 -8984.763,E2 -8984.763} C_VEL
LIN {X 0,Y 441.648,Z 608.183,A -85,B 0,C 180,E1 -8985.367,E2 -8985.367} C_VEL
LIN {X 0,Y 441.114,Z 620.647,A -85,B 0,C 180,E1 -8986.173,E2 -8986.173} C_VEL
LIN {X 0,Y 440.685,Z 631.8,A -85,B 0,C 180,E1 -8987.099,E2 -8987.099} C_VEL
LIN {X 0,Y 440.078,Z 642.888,A -85,B 0,C 180,E1 -8988.251,E2 -8988.251} C_VEL
LIN {X 0,Y 439.631,Z 651.862,A -85,B 0,C 180,E1 -8989.406,E2 -8989.406} C_VEL
LIN {X 0,Y 439.202,Z 660.558,A -85,B 0,C 180,E1 -8990.792,E2 -8990.792} C_VEL
LIN {X 0,Y 438.799,Z 667.56,A -85,B 0,C 180,E1 -8992.175,E2 -8992.175} C_VEL
LIN {X 0,Y 438.614,Z 673.099,A -85,B 0,C 180,E1 -8993.56,E2 -8993.56} C_VEL
LIN {X 0,Y 438.47,Z 677.416,A -85,B 0,C 180,E1 -8994.942,E2 -8994.942} C_VEL
LIN {X 0,Y 438.383,Z 680.633,A -85,B 0,C 180,E1 -8996.323,E2 -8996.323} C_VEL
LIN {X 0,Y 438.389,Z 682.221,A -85,B 0,C 180,E1 -8997.243,E2 -8997.243} C_VEL
LIN {X 0,Y 438.3,Z 683.363,A -85,B 0,C 180,E1 -8998.162,E2 -8998.162} C_VEL
LIN {X 0,Y 438.255,Z 684.065,A -85,B 0,C 180,E1 -8999.081,E2 -8999.081} C_VEL
LIN {X 0,Y 438.253,Z 684.37,A -85,B 0,C 180,E1 -9000,E2 -9000} C_VEL
LIN {X 0,Y 438.255,Z 684.241,A -85,B 0,C 180,E1 -9000.919,E2 -9000.919} C_VEL
LIN {X 0,Y 438.301,Z 683.671,A -85,B 0,C 180,E1 -9001.838,E2 -9001.838} C_VEL
LIN {X 0,Y 438.391,Z 682.702,A -85,B 0,C 180,E1 -9002.757,E2 -9002.757} C_VEL
LIN {X 0,Y 438.405,Z 681.296,A -85,B 0,C 180,E1 -9003.676,E2 -9003.676} C_VEL
LIN {X 0,Y 438.472,Z 678.336,A -85,B 0,C 180,E1 -9005.058,E2 -9005.058} C_VEL
LIN {X 0,Y 438.643,Z 674.285,A -85,B 0,C 180,E1 -9006.44,E2 -9006.44} C_VEL
LIN {X 0,Y 438.923,Z 668.052,A -85,B 0,C 180,E1 -9008.054,E2 -9008.054} C_VEL
LIN {X 0,Y 439.32,Z 661.164,A -85,B 0,C 180,E1 -9009.438,E2 -9009.438} C_VEL
LIN {X 0,Y 439.821,Z 652.575,A -85,B 0,C 180,E1 -9010.822,E2 -9010.822} C_VEL
LIN {X 0,Y 440.352,Z 642.741,A -85,B 0,C 180,E1 -9012.092,E2 -9012.092} C_VEL
LIN {X 0,Y 440.939,Z 632.464,A -85,B 0,C 180,E1 -9013.162,E2 -9013.162} C_VEL
LIN {X 0,Y 441.417,Z 621.914,A -85,B 0,C 180,E1 -9014.052,E2 -9014.052} C_VEL
LIN {X 0,Y 441.976,Z 609.734,A -85,B 0,C 180,E1 -9014.857,E2 -9014.857} C_VEL
LIN {X 0,Y 442.449,Z 598.427,A -85,B 0,C 180,E1 -9015.43,E2 -9015.43} C_VEL
LIN {X 0,Y 442.807,Z 585.802,A -85,B 0,C 180,E1 -9015.89,E2 -9015.89} C_VEL
LIN {X 0,Y 443.136,Z 570.565,A -85,B 0,C 180,E1 -9016.232,E2 -9016.232} C_VEL
LIN {X 0,Y 444.563,Z 490.773,A -85,B 0,C 180,E1 -9017.836,E2 -9017.836} C_VEL
LIN {X 0,Y 443.978,Z 484.506,A -85,B 0,C 180,E1 -9018.007,E2 -9018.007} C_VEL
LIN {X 0,Y 441.717,Z 472.723,A -85,B 0,C 180,E1 -9018.401,E2 -9018.401} C_VEL
LIN {X 0,Y 442.499,Z 452.639,A -85,B 0,C 180,E1 -9021.671,E2 -9021.671} C_VEL
LIN {X 0,Y 443.057,Z 436.03,A -85,B 0,C 180,E1 -9024.357,E2 -9024.357} C_VEL
LIN {X 0,Y 441.479,Z 426.977,A -85,B 0,C 180,E1 -9025.962,E2 -9025.962} C_VEL
LIN {X 0,Y 439.392,Z 418.755,A -85,B 0,C 180,E1 -9027.507,E2 -9027.507} C_VEL
LIN {X 0,Y 439.362,Z 418.76,A -85,B 0,C 180,E1 -9030.789,E2 -9030.789} C_VEL
LIN {X 0,Y 439.389,Z 418.754,A -85,B 0,C 180,E1 -9034.044,E2 -9034.044} C_VEL
LIN {X 0,Y 439.349,Z 418.757,A -85,B 0,C 180,E1 -9036.887,E2 -9036.887} C_VEL
LIN {X 0,Y 439.404,Z 418.75,A -85,B 0,C 180,E1 -9039.849,E2 -9039.849} C_VEL
LIN {X 0,Y 439.385,Z 418.754,A -85,B 0,C 180,E1 -9042.627,E2 -9042.627} C_VEL
LIN {X 0,Y 439.404,Z 418.751,A -85,B 0,C 180,E1 -9045.271,E2 -9045.271} C_VEL
LIN {X 0,Y 439.391,Z 418.752,A -85,B 0,C 180,E1 -9048.743,E2 -9048.743} C_VEL
LIN {X 0,Y 439.375,Z 418.753,A -85,B 0,C 180,E1 -9051.608,E2 -9051.608} C_VEL
LIN {X 0,Y 439.4,Z 418.751,A -85,B 0,C 180,E1 -9054.844,E2 -9054.844} C_VEL
LIN {X 0,Y 439.374,Z 418.754,A -85,B 0,C 180,E1 -9058.14,E2 -9058.14} C_VEL
LIN {X 0,Y 439.41,Z 418.817,A -85,B 0,C 180,E1 -9060.349,E2 -9060.349} C_VEL
LIN {X 0,Y 442.852,Z 434.973,A -85,B 0,C 180,E1 -9063.178,E2 -9063.178} C_VEL
LIN {X 0,Y 443.012,Z 439.254,A -85,B 0,C 180,E1 -9063.881,E2 -9063.881} C_VEL
LIN {X 0,Y 442.015,Z 456.258,A -85,B 0,C 180,E1 -9066.578,E2 -9066.578} C_VEL
LIN {X 0,Y 441.176,Z 474.759,A -85,B 0,C 180,E1 -9069.484,E2 -9069.484} C_VEL
LIN {X 0,Y 440.44,Z 490.762,A -85,B 0,C 180,E1 -9071.973,E2 -9071.973} C_VEL
LIN {X 0,Y 443.549,Z 516.811,A -85,B 0,C 180,E1 -9072.608,E2 -9072.608} C_VEL
LIN {X 0,Y 442.629,Z 604.091,A -85,B 0,C 180,E1 -9074.045,E2 -9074.045} C_VEL
LIN {X 0,Y 442.357,Z 617.038,A -85,B 0,C 180,E1 -9074.419,E2 -9074.419} C_VEL
LIN {X 0,Y 441.78,Z 630.581,A -85,B 0,C 180,E1 -9075.018,E2 -9075.018} C_VEL
LIN {X 0,Y 441.252,Z 641.924,A -85,B 0,C 180,E1 -9075.707,E2 -9075.707} C_VEL
LIN {X 0,Y 440.678,Z 653.402,A -85,B 0,C 180,E1 -9076.616,E2 -9076.616} C_VEL
LIN {X 0,Y 440.1,Z 663.982,A -85,B 0,C 180,E1 -9077.667,E2 -9077.667} C_VEL
LIN {X 0,Y 439.625,Z 672.493,A -85,B 0,C 180,E1 -9078.707,E2 -9078.707} C_VEL
LIN {X 0,Y 439.178,Z 680.314,A -85,B 0,C 180,E1 -9079.861,E2 -9079.861} C_VEL
LIN {X 0,Y 438.84,Z 687.926,A -85,B 0,C 180,E1 -9081.249,E2 -9081.249} C_VEL
LIN {X 0,Y 438.584,Z 694.034,A -85,B 0,C 180,E1 -9082.635,E2 -9082.635} C_VEL
LIN {X 0,Y 438.418,Z 698.598,A -85,B 0,C 180,E1 -9083.936,E2 -9083.936} C_VEL
LIN {X 0,Y 438.392,Z 702.537,A -85,B 0,C 180,E1 -9085.402,E2 -9085.402} C_VEL
LIN {X 0,Y 438.381,Z 704.434,A -85,B 0,C 180,E1 -9086.323,E2 -9086.323} C_VEL
LIN {X 0,Y 438.415,Z 705.867,A -85,B 0,C 180,E1 -9087.243,E2 -9087.243} C_VEL
LIN {X 0,Y 438.315,Z 707.49,A -85,B 0,C 180,E1 -9089.081,E2 -9089.081} C_VEL
LIN {X 0,Y 438.326,Z 707.712,A -85,B 0,C 180,E1 -9090,E2 -9090} C_VEL
LIN {X 0,Y 438.315,Z 707.49,A -85,B 0,C 180,E1 -9090.919,E2 -9090.919} C_VEL
LIN {X 0,Y 438.418,Z 705.866,A -85,B 0,C 180,E1 -9092.756,E2 -9092.756} C_VEL
LIN {X 0,Y 438.391,Z 704.432,A -85,B 0,C 180,E1 -9093.677,E2 -9093.677} C_VEL
LIN {X 0,Y 438.44,Z 701.449,A -85,B 0,C 180,E1 -9095.058,E2 -9095.058} C_VEL
LIN {X 0,Y 438.506,Z 697.397,A -85,B 0,C 180,E1 -9096.442,E2 -9096.442} C_VEL
LIN {X 0,Y 438.692,Z 691.146,A -85,B 0,C 180,E1 -9098.058,E2 -9098.058} C_VEL
LIN {X 0,Y 439.019,Z 684.324,A -85,B 0,C 180,E1 -9099.444,E2 -9099.444} C_VEL
LIN {X 0,Y 439.337,Z 677.337,A -85,B 0,C 180,E1 -9100.601,E2 -9100.601} C_VEL
LIN {X 0,Y 439.852,Z 668.892,A -85,B 0,C 180,E1 -9101.755,E2 -9101.755} C_VEL
LIN {X 0,Y 440.424,Z 658.429,A -85,B 0,C 180,E1 -9102.909,E2 -9102.909} C_VEL
LIN {X 0,Y 440.947,Z 648.05,A -85,B 0,C 180,E1 -9103.832,E2 -9103.832} C_VEL
LIN {X 0,Y 441.534,Z 636.592,A -85,B 0,C 180,E1 -9104.637,E2 -9104.637} C_VEL
LIN {X 0,Y 442.074,Z 624.667,A -85,B 0,C 180,E1 -9105.266,E2 -9105.266} C_VEL
LIN {X 0,Y 442.52,Z 611.745,A -85,B 0,C 180,E1 -9105.752,E2 -9105.752} C_VEL
LIN {X 0,Y 442.782,Z 599.478,A -85,B 0,C 180,E1 -9106.038,E2 -9106.038} C_VEL
LIN {X 0,Y 443.224,Z 566.686,A -85,B 0,C 180,E1 -9106.608,E2 -9106.608} C_VEL
LIN {X 0,Y 443.894,Z 515.328,A -85,B 0,C 180,E1 -9107.651,E2 -9107.651} C_VEL
LIN {X 0,Y 441.216,Z 491.383,A -85,B 0,C 180,E1 -9108.311,E2 -9108.311} C_VEL
LIN {X 0,Y 440.372,Z 485.948,A -85,B 0,C 180,E1 -9108.481,E2 -9108.481} C_VEL
LIN {X 0,Y 441.37,Z 465.577,A -85,B 0,C 180,E1 -9111.729,E2 -9111.729} C_VEL
LIN {X 0,Y 442.6,Z 444.693,A -85,B 0,C 180,E1 -9115.163,E2 -9115.163} C_VEL
LIN {X 0,Y 443.16,Z 436.362,A -85,B 0,C 180,E1 -9116.575,E2 -9116.575} C_VEL
LIN {X 0,Y 441.208,Z 426.158,A -85,B 0,C 180,E1 -9118.547,E2 -9118.547} C_VEL
LIN {X 0,Y 439.383,Z 418.76,A -85,B 0,C 180,E1 -9120.094,E2 -9120.094} C_VEL
LIN {X 0,Y 439.375,Z 418.756,A -85,B 0,C 180,E1 -9122.946,E2 -9122.946} C_VEL
LIN {X 0,Y 439.374,Z 418.755,A -85,B 0,C 180,E1 -9126.287,E2 -9126.287} C_VEL
LIN {X 0,Y 439.404,Z 418.753,A -85,B 0,C 180,E1 -9129.849,E2 -9129.849} C_VEL
LIN {X 0,Y 439.372,Z 418.753,A -85,B 0,C 180,E1 -9132.625,E2 -9132.625} C_VEL
LIN {X 0,Y 439.403,Z 418.752,A -85,B 0,C 180,E1 -9135.271,E2 -9135.271} C_VEL
LIN {X 0,Y 439.391,Z 418.752,A -85,B 0,C 180,E1 -9138.743,E2 -9138.743} C_VEL
LIN {X 0,Y 439.379,Z 418.754,A -85,B 0,C 180,E1 -9141.607,E2 -9141.607} C_VEL
LIN {X 0,Y 439.402,Z 418.752,A -85,B 0,C 180,E1 -9144.844,E2 -9144.844} C_VEL
LIN {X 0,Y 439.376,Z 418.754,A -85,B 0,C 180,E1 -9148.14,E2 -9148.14} C_VEL
LIN {X 0,Y 439.435,Z 418.748,A -85,B 0,C 180,E1 -9151.598,E2 -9151.598} C_VEL
LIN {X 0,Y 439.4,Z 418.755,A -85,B 0,C 180,E1 -9154.415,E2 -9154.415} C_VEL
LIN {X 0,Y 439.367,Z 418.759,A -85,B 0,C 180,E1 -9157.425,E2 -9157.425} C_VEL
LIN {X 0,Y 439.443,Z 418.749,A -85,B 0,C 180,E1 -9160.663,E2 -9160.663} C_VEL
LIN {X 0,Y 439.414,Z 418.752,A -85,B 0,C 180,E1 -9161.621,E2 -9161.621} C_VEL
LIN {X 0,Y 440.444,Z 421.623,A -85,B 0,C 180,E1 -9161.752,E2 -9161.752} C_VEL
LIN {X 0,Y 444.931,Z 432.429,A -85,B 0,C 180,E1 -9162.249,E2 -9162.249} C_VEL
LIN {X 0,Y 443.511,Z 503.815,A -85,B 0,C 180,E1 -9163.723,E2 -9163.723} C_VEL
LIN {X 0,Y 443.252,Z 523.622,A -85,B 0,C 180,E1 -9164.156,E2 -9164.156} C_VEL
LIN {X 0,Y 442.962,Z 535.744,A -85,B 0,C 180,E1 -9164.588,E2 -9164.588} C_VEL
LIN {X 0,Y 442.679,Z 547.243,A -85,B 0,C 180,E1 -9165.167,E2 -9165.167} C_VEL
LIN {X 0,Y 442.169,Z 559.526,A -85,B 0,C 180,E1 -9165.981,E2 -9165.981} C_VEL
LIN {X 0,Y 441.651,Z 570.342,A -85,B 0,C 180,E1 -9166.894,E2 -9166.894} C_VEL
LIN {X 0,Y 441.222,Z 579.19,A -85,B 0,C 180,E1 -9167.816,E2 -9167.816} C_VEL
LIN {X 0,Y 440.682,Z 588.261,A -85,B 0,C 180,E1 -9168.967,E2 -9168.967} C_VEL
LIN {X 0,Y 440.14,Z 597.083,A -85,B 0,C 180,E1 -9170.348,E2 -9170.348} C_VEL
LIN {X 0,Y 439.758,Z 604.135,A -85,B 0,C 180,E1 -9171.73,E2 -9171.73} C_VEL
LIN {X 0,Y 439.377,Z 610.172,A -85,B 0,C 180,E1 -9173.247,E2 -9173.247} C_VEL
LIN {X 0,Y 439.081,Z 614.046,A -85,B 0,C 180,E1 -9174.489,E2 -9174.489} C_VEL
LIN {X 0,Y 439.092,Z 616.296,A -85,B 0,C 180,E1 -9175.41,E2 -9175.41} C_VEL
LIN {X 0,Y 438.887,Z 618.136,A -85,B 0,C 180,E1 -9176.328,E2 -9176.328} C_VEL
LIN {X 0,Y 438.673,Z 619.503,A -85,B 0,C 180,E1 -9177.245,E2 -9177.245} C_VEL
LIN {X 0,Y 438.552,Z 620.436,A -85,B 0,C 180,E1 -9178.163,E2 -9178.163} C_VEL
LIN {X 0,Y 438.503,Z 620.964,A -85,B 0,C 180,E1 -9179.082,E2 -9179.082} C_VEL
LIN {X 0,Y 438.482,Z 621.079,A -85,B 0,C 180,E1 -9180,E2 -9180} C_VEL
LIN {X 0,Y 438.478,Z 620.745,A -85,B 0,C 180,E1 -9180.918,E2 -9180.918} C_VEL
LIN {X 0,Y 438.523,Z 620.01,A -85,B 0,C 180,E1 -9181.837,E2 -9181.837} C_VEL
LIN {X 0,Y 438.662,Z 618.87,A -85,B 0,C 180,E1 -9182.755,E2 -9182.755} C_VEL
LIN {X 0,Y 438.902,Z 616.326,A -85,B 0,C 180,E1 -9184.132,E2 -9184.132} C_VEL
LIN {X 0,Y 438.955,Z 612.78,A -85,B 0,C 180,E1 -9185.513,E2 -9185.513} C_VEL
LIN {X 0,Y 439.15,Z 608.281,A -85,B 0,C 180,E1 -9186.846,E2 -9186.846} C_VEL
LIN {X 0,Y 439.392,Z 602.157,A -85,B 0,C 180,E1 -9188.277,E2 -9188.277} C_VEL
LIN {X 0,Y 439.832,Z 594.694,A -85,B 0,C 180,E1 -9189.659,E2 -9189.659} C_VEL
LIN {X 0,Y 440.297,Z 585.431,A -85,B 0,C 180,E1 -9191.043,E2 -9191.043} C_VEL
LIN {X 0,Y 440.8,Z 575.798,A -85,B 0,C 180,E1 -9192.196,E2 -9192.196} C_VEL
LIN {X 0,Y 441.266,Z 565.574,A -85,B 0,C 180,E1 -9193.193,E2 -9193.193} C_VEL
LIN {X 0,Y 441.653,Z 554.823,A -85,B 0,C 180,E1 -9194.044,E2 -9194.044} C_VEL
LIN {X 0,Y 442,Z 542.687,A -85,B 0,C 180,E1 -9194.797,E2 -9194.797} C_VEL
LIN {X 0,Y 442.415,Z 529.375,A -85,B 0,C 180,E1 -9195.402,E2 -9195.402} C_VEL
LIN {X 0,Y 442.647,Z 516.279,A -85,B 0,C 180,E1 -9195.807,E2 -9195.807} C_VEL
LIN {X 0,Y 443.757,Z 431.596,A -85,B 0,C 180,E1 -9197.399,E2 -9197.399} C_VEL
LIN {X 0,Y 439.438,Z 418.752,A -85,B 0,C 180,E1 -9197.822,E2 -9197.822} C_VEL
LIN {X 0,Y 439.39,Z 418.754,A -85,B 0,C 180,E1 -9200.603,E2 -9200.603} C_VEL
LIN {X 0,Y 439.385,Z 418.752,A -85,B 0,C 180,E1 -9203.571,E2 -9203.571} C_VEL
LIN {X 0,Y 439.421,Z 418.746,A -85,B 0,C 180,E1 -9206.604,E2 -9206.604} C_VEL
LIN {X 0,Y 439.385,Z 418.752,A -85,B 0,C 180,E1 -9209.726,E2 -9209.726} C_VEL
LIN {X 0,Y 439.375,Z 418.743,A -85,B 0,C 180,E1 -9212.946,E2 -9212.946} C_VEL
LIN {X 0,Y 439.376,Z 418.751,A -85,B 0,C 180,E1 -9216.287,E2 -9216.287} C_VEL
LIN {X 0,Y 439.404,Z 418.741,A -85,B 0,C 180,E1 -9219.849,E2 -9219.849} C_VEL
LIN {X 0,Y 439.385,Z 418.754,A -85,B 0,C 180,E1 -9222.627,E2 -9222.627} C_VEL
LIN {X 0,Y 439.404,Z 418.742,A -85,B 0,C 180,E1 -9225.271,E2 -9225.271} C_VEL
LIN {X 0,Y 439.391,Z 418.752,A -85,B 0,C 180,E1 -9228.743,E2 -9228.743} C_VEL
LIN {X 0,Y 439.375,Z 418.753,A -85,B 0,C 180,E1 -9231.608,E2 -9231.608} C_VEL
LIN {X 0,Y 439.401,Z 418.752,A -85,B 0,C 180,E1 -9234.844,E2 -9234.844} C_VEL
LIN {X 0,Y 439.375,Z 418.755,A -85,B 0,C 180,E1 -9238.14,E2 -9238.14} C_VEL
LIN {X 0,Y 439.402,Z 418.755,A -85,B 0,C 180,E1 -9241.606,E2 -9241.606} C_VEL
LIN {X 0,Y 439.396,Z 418.799,A -85,B 0,C 180,E1 -9243.041,E2 -9243.041} C_VEL
LIN {X 0,Y 442.256,Z 432.663,A -85,B 0,C 180,E1 -9245.596,E2 -9245.596} C_VEL
LIN {X 0,Y 442.222,Z 440.679,A -85,B 0,C 180,E1 -9246.978,E2 -9246.978} C_VEL
LIN {X 0,Y 441.406,Z 461.678,A -85,B 0,C 180,E1 -9250.466,E2 -9250.466} C_VEL
LIN {X 0,Y 441.157,Z 471.125,A -85,B 0,C 180,E1 -9251.942,E2 -9251.942} C_VEL
LIN {X 0,Y 441.474,Z 473.037,A -85,B 0,C 180,E1 -9251.994,E2 -9251.994} C_VEL
LIN {X 0,Y 441.741,Z 478.883,A -85,B 0,C 180,E1 -9252.104,E2 -9252.104} C_VEL
LIN {X 0,Y 440.943,Z 484.768,A -85,B 0,C 180,E1 -9252.17,E2 -9252.17} C_VEL
LIN {X 0,Y 437.562,Z 500.475,A -85,B 0,C 180,E1 -9252.293,E2 -9252.293} C_VEL
LIN {X 0,Y 437.273,Z 504.461,A -85,B 0,C 180,E1 -9252.349,E2 -9252.349} C_VEL
LIN {X 0,Y 436.459,Z 580.836,A -85,B 0,C 180,E1 -9253.633,E2 -9253.633} C_VEL
LIN {X 0,Y 436.157,Z 594.342,A -85,B 0,C 180,E1 -9254.042,E2 -9254.042} C_VEL
LIN {X 0,Y 435.628,Z 606.917,A -85,B 0,C 180,E1 -9254.622,E2 -9254.622} C_VEL
LIN {X 0,Y 435.041,Z 619.036,A -85,B 0,C 180,E1 -9255.379,E2 -9255.379} C_VEL
LIN {X 0,Y 434.502,Z 629.639,A -85,B 0,C 180,E1 -9256.234,E2 -9256.234} C_VEL
LIN {X 0,Y 433.915,Z 639.734,A -85,B 0,C 180,E1 -9257.251,E2 -9257.251} C_VEL
LIN {X 0,Y 433.122,Z 650.061,A -85,B 0,C 180,E1 -9258.535,E2 -9258.535} C_VEL
LIN {X 0,Y 432.541,Z 659.019,A -85,B 0,C 180,E1 -9259.941,E2 -9259.941} C_VEL
LIN {X 0,Y 432.053,Z 666.209,A -85,B 0,C 180,E1 -9261.346,E2 -9261.346} C_VEL
LIN {X 0,Y 431.673,Z 672.808,A -85,B 0,C 180,E1 -9262.987,E2 -9262.987} C_VEL
LIN {X 0,Y 431.529,Z 677.138,A -85,B 0,C 180,E1 -9264.392,E2 -9264.392} C_VEL
LIN {X 0,Y 431.343,Z 679.421,A -85,B 0,C 180,E1 -9265.327,E2 -9265.327} C_VEL
LIN {X 0,Y 431.312,Z 681.28,A -85,B 0,C 180,E1 -9266.263,E2 -9266.263} C_VEL
LIN {X 0,Y 431.323,Z 682.701,A -85,B 0,C 180,E1 -9267.198,E2 -9267.198} C_VEL
LIN {X 0,Y 431.172,Z 684.315,A -85,B 0,C 180,E1 -9269.066,E2 -9269.066} C_VEL
LIN {X 0,Y 431.168,Z 684.551,A -85,B 0,C 180,E1 -9270,E2 -9270} C_VEL
LIN {X 0,Y 431.172,Z 684.362,A -85,B 0,C 180,E1 -9270.934,E2 -9270.934} C_VEL
LIN {X 0,Y 431.323,Z 682.809,A -85,B 0,C 180,E1 -9272.802,E2 -9272.802} C_VEL
LIN {X 0,Y 431.311,Z 681.448,A -85,B 0,C 180,E1 -9273.737,E2 -9273.737} C_VEL
LIN {X 0,Y 431.424,Z 678.581,A -85,B 0,C 180,E1 -9275.14,E2 -9275.14} C_VEL
LIN {X 0,Y 431.614,Z 674.339,A -85,B 0,C 180,E1 -9276.65,E2 -9276.65} C_VEL
LIN {X 0,Y 431.872,Z 669.639,A -85,B 0,C 180,E1 -9277.951,E2 -9277.951} C_VEL
LIN {X 0,Y 432.284,Z 663.275,A -85,B 0,C 180,E1 -9279.357,E2 -9279.357} C_VEL
LIN {X 0,Y 432.819,Z 655.368,A -85,B 0,C 180,E1 -9280.762,E2 -9280.762} C_VEL
LIN {X 0,Y 433.323,Z 647.292,A -85,B 0,C 180,E1 -9281.934,E2 -9281.934} C_VEL
LIN {X 0,Y 434.051,Z 637.367,A -85,B 0,C 180,E1 -9283.102,E2 -9283.102} C_VEL
LIN {X 0,Y 434.655,Z 626.216,A -85,B 0,C 180,E1 -9284.156,E2 -9284.156} C_VEL
LIN {X 0,Y 435.258,Z 615.304,A -85,B 0,C 180,E1 -9284.972,E2 -9284.972} C_VEL
LIN {X 0,Y 435.841,Z 603.048,A -85,B 0,C 180,E1 -9285.67,E2 -9285.67} C_VEL
LIN {X 0,Y 436.295,Z 589.496,A -85,B 0,C 180,E1 -9286.223,E2 -9286.223} C_VEL
LIN {X 0,Y 436.6,Z 576.887,A -85,B 0,C 180,E1 -9286.542,E2 -9286.542} C_VEL
LIN {X 0,Y 437.334,Z 488.969,A -85,B 0,C 180,E1 -9288.006,E2 -9288.006} C_VEL
LIN {X 0,Y 434.256,Z 471.268,A -85,B 0,C 180,E1 -9288.445,E2 -9288.445} C_VEL
LIN {X 0,Y 434.763,Z 454.898,A -85,B 0,C 180,E1 -9291.08,E2 -9291.08} C_VEL
LIN {X 0,Y 435.514,Z 437.486,A -85,B 0,C 180,E1 -9294.046,E2 -9294.046} C_VEL
LIN {X 0,Y 435.14,Z 433.056,A -85,B 0,C 180,E1 -9294.83,E2 -9294.83} C_VEL
LIN {X 0,Y 432.329,Z 419.636,A -85,B 0,C 180,E1 -9297.338,E2 -9297.338} C_VEL
LIN {X 0,Y 432.348,Z 419.63,A -85,B 0,C 180,E1 -9300.51,E2 -9300.51} C_VEL
LIN {X 0,Y 432.362,Z 419.631,A -85,B 0,C 180,E1 -9304.003,E2 -9304.003} C_VEL
LIN {X 0,Y 432.323,Z 419.634,A -85,B 0,C 180,E1 -9307.197,E2 -9307.197} C_VEL
LIN {X 0,Y 432.335,Z 419.625,A -85,B 0,C 180,E1 -9310.179,E2 -9310.179} C_VEL
LIN {X 0,Y 432.32,Z 419.633,A -85,B 0,C 180,E1 -9313.061,E2 -9313.061} C_VEL
LIN {X 0,Y 432.343,Z 419.631,A -85,B 0,C 180,E1 -9315.664,E2 -9315.664} C_VEL
LIN {X 0,Y 432.336,Z 419.625,A -85,B 0,C 180,E1 -9318.398,E2 -9318.398} C_VEL
LIN {X 0,Y 432.34,Z 419.628,A -85,B 0,C 180,E1 -9321.85,E2 -9321.85} C_VEL
LIN {X 0,Y 432.342,Z 419.628,A -85,B 0,C 180,E1 -9325.323,E2 -9325.323} C_VEL
LIN {X 0,Y 432.323,Z 419.636,A -85,B 0,C 180,E1 -9328.654,E2 -9328.654} C_VEL
LIN {X 0,Y 432.341,Z 419.632,A -85,B 0,C 180,E1 -9331.874,E2 -9331.874} C_VEL
LIN {X 0,Y 432.373,Z 419.69,A -85,B 0,C 180,E1 -9332.958,E2 -9332.958} C_VEL
LIN {X 0,Y 435.112,Z 433.342,A -85,B 0,C 180,E1 -9335.423,E2 -9335.423} C_VEL
LIN {X 0,Y 435.383,Z 439.244,A -85,B 0,C 180,E1 -9336.436,E2 -9336.436} C_VEL
LIN {X 0,Y 434.587,Z 459.652,A -85,B 0,C 180,E1 -9339.858,E2 -9339.858} C_VEL
LIN {X 0,Y 434.065,Z 471.733,A -85,B 0,C 180,E1 -9341.864,E2 -9341.864} C_VEL
LIN {X 0,Y 436.868,Z 489.232,A -85,B 0,C 180,E1 -9342.32,E2 -9342.32} C_VEL
LIN {X 0,Y 435.57,Z 581.951,A -85,B 0,C 180,E1 -9344.11,E2 -9344.11} C_VEL
LIN {X 0,Y 435.132,Z 595.747,A -85,B 0,C 180,E1 -9344.574,E2 -9344.574} C_VEL
LIN {X 0,Y 434.694,Z 608.292,A -85,B 0,C 180,E1 -9345.188,E2 -9345.188} C_VEL
LIN {X 0,Y 434.128,Z 621.271,A -85,B 0,C 180,E1 -9346.043,E2 -9346.043} C_VEL
LIN {X 0,Y 433.653,Z 632.546,A -85,B 0,C 180,E1 -9347.005,E2 -9347.005} C_VEL
LIN {X 0,Y 433.074,Z 642.537,A -85,B 0,C 180,E1 -9348.059,E2 -9348.059} C_VEL
LIN {X 0,Y 432.613,Z 651.64,A -85,B 0,C 180,E1 -9349.232,E2 -9349.232} C_VEL
LIN {X 0,Y 432.137,Z 660.419,A -85,B 0,C 180,E1 -9350.64,E2 -9350.64} C_VEL
LIN {X 0,Y 431.76,Z 667.503,A -85,B 0,C 180,E1 -9352.047,E2 -9352.047} C_VEL
LIN {X 0,Y 431.563,Z 673.11,A -85,B 0,C 180,E1 -9353.454,E2 -9353.454} C_VEL
LIN {X 0,Y 431.41,Z 677.477,A -85,B 0,C 180,E1 -9354.859,E2 -9354.859} C_VEL
LIN {X 0,Y 431.284,Z 680.736,A -85,B 0,C 180,E1 -9356.263,E2 -9356.263} C_VEL
LIN {X 0,Y 431.301,Z 682.345,A -85,B 0,C 180,E1 -9357.198,E2 -9357.198} C_VEL
LIN {X 0,Y 431.225,Z 683.519,A -85,B 0,C 180,E1 -9358.132,E2 -9358.132} C_VEL
LIN {X 0,Y 431.172,Z 684.238,A -85,B 0,C 180,E1 -9359.066,E2 -9359.066} C_VEL
LIN {X 0,Y 431.168,Z 684.559,A -85,B 0,C 180,E1 -9360,E2 -9360} C_VEL
LIN {X 0,Y 431.172,Z 684.456,A -85,B 0,C 180,E1 -9360.934,E2 -9360.934} C_VEL
LIN {X 0,Y 431.225,Z 683.898,A -85,B 0,C 180,E1 -9361.868,E2 -9361.868} C_VEL
LIN {X 0,Y 431.322,Z 682.938,A -85,B 0,C 180,E1 -9362.802,E2 -9362.802} C_VEL
LIN {X 0,Y 431.312,Z 681.552,A -85,B 0,C 180,E1 -9363.737,E2 -9363.737} C_VEL
LIN {X 0,Y 431.418,Z 678.606,A -85,B 0,C 180,E1 -9365.14,E2 -9365.14} C_VEL
LIN {X 0,Y 431.582,Z 674.343,A -85,B 0,C 180,E1 -9366.614,E2 -9366.614} C_VEL
LIN {X 0,Y 431.903,Z 668.357,A -85,B 0,C 180,E1 -9368.186,E2 -9368.186} C_VEL
LIN {X 0,Y 432.31,Z 661.494,A -85,B 0,C 180,E1 -9369.592,E2 -9369.592} C_VEL
LIN {X 0,Y 432.86,Z 652.92,A -85,B 0,C 180,E1 -9370.998,E2 -9370.998} C_VEL
LIN {X 0,Y 433.353,Z 644.137,A -85,B 0,C 180,E1 -9372.171,E2 -9372.171} C_VEL
LIN {X 0,Y 434.028,Z 633.127,A -85,B 0,C 180,E1 -9373.352,E2 -9373.352} C_VEL
LIN {X 0,Y 434.551,Z 622.417,A -85,B 0,C 180,E1 -9374.279,E2 -9374.279} C_VEL
LIN {X 0,Y 435.152,Z 610.34,A -85,B 0,C 180,E1 -9375.096,E2 -9375.096} C_VEL
LIN {X 0,Y 435.702,Z 597.905,A -85,B 0,C 180,E1 -9375.735,E2 -9375.735} C_VEL
LIN {X 0,Y 436.121,Z 584.023,A -85,B 0,C 180,E1 -9376.23,E2 -9376.23} C_VEL
LIN {X 0,Y 438.032,Z 490.168,A -85,B 0,C 180,E1 -9378.202,E2 -9378.202} C_VEL
LIN {X 0,Y 435.657,Z 476.285,A -85,B 0,C 180,E1 -9378.654,E2 -9378.654} C_VEL
LIN {X 0,Y 434.961,Z 472.802,A -85,B 0,C 180,E1 -9378.806,E2 -9378.806} C_VEL
LIN {X 0,Y 435.717,Z 454.776,A -85,B 0,C 180,E1 -9381.776,E2 -9381.776} C_VEL
LIN {X 0,Y 436.352,Z 438.161,A -85,B 0,C 180,E1 -9384.503,E2 -9384.503} C_VEL
LIN {X 0,Y 435.154,Z 430.627,A -85,B 0,C 180,E1 -9385.853,E2 -9385.853} C_VEL
LIN {X 0,Y 432.343,Z 419.635,A -85,B 0,C 180,E1 -9387.961,E2 -9387.961} C_VEL
LIN {X 0,Y 432.323,Z 419.637,A -85,B 0,C 180,E1 -9391.346,E2 -9391.346} C_VEL
LIN {X 0,Y 432.341,Z 419.632,A -85,B 0,C 180,E1 -9394.677,E2 -9394.677} C_VEL
LIN {X 0,Y 432.34,Z 419.629,A -85,B 0,C 180,E1 -9398.15,E2 -9398.15} C_VEL
LIN {X 0,Y 432.335,Z 419.631,A -85,B 0,C 180,E1 -9401.602,E2 -9401.602} C_VEL
LIN {X 0,Y 432.336,Z 419.632,A -85,B 0,C 180,E1 -9404.347,E2 -9404.347} C_VEL
LIN {X 0,Y 432.323,Z 419.633,A -85,B 0,C 180,E1 -9407.016,E2 -9407.016} C_VEL
LIN {X 0,Y 432.338,Z 419.63,A -85,B 0,C 180,E1 -9409.82,E2 -9409.82} C_VEL
LIN {X 0,Y 432.307,Z 419.634,A -85,B 0,C 180,E1 -9413.022,E2 -9413.022} C_VEL
LIN {X 0,Y 432.361,Z 419.628,A -85,B 0,C 180,E1 -9415.997,E2 -9415.997} C_VEL
LIN {X 0,Y 432.348,Z 419.631,A -85,B 0,C 180,E1 -9419.49,E2 -9419.49} C_VEL
LIN {X 0,Y 432.379,Z 419.845,A -85,B 0,C 180,E1 -9420.146,E2 -9420.146} C_VEL
LIN {X 0,Y 436.009,Z 436.845,A -85,B 0,C 180,E1 -9423.171,E2 -9423.171} C_VEL
LIN {X 0,Y 435.827,Z 444.777,A -85,B 0,C 180,E1 -9424.468,E2 -9424.468} C_VEL
LIN {X 0,Y 434.58,Z 466.259,A -85,B 0,C 180,E1 -9427.914,E2 -9427.914} C_VEL
LIN {X 0,Y 433.634,Z 486.233,A -85,B 0,C 180,E1 -9431.086,E2 -9431.086} C_VEL
LIN {X 0,Y 433.494,Z 489.523,A -85,B 0,C 180,E1 -9431.569,E2 -9431.569} C_VEL
LIN {X 0,Y 436.337,Z 514.18,A -85,B 0,C 180,E1 -9432.285,E2 -9432.285} C_VEL
LIN {X 0,Y 436.68,Z 521.969,A -85,B 0,C 180,E1 -9432.43,E2 -9432.43} C_VEL
LIN {X 0,Y 435.846,Z 602.55,A -85,B 0,C 180,E1 -9433.76,E2 -9433.76} C_VEL
LIN {X 0,Y 435.56,Z 615.322,A -85,B 0,C 180,E1 -9434.109,E2 -9434.109} C_VEL
LIN {X 0,Y 435.041,Z 628.187,A -85,B 0,C 180,E1 -9434.661,E2 -9434.661} C_VEL
LIN {X 0,Y 434.447,Z 640.022,A -85,B 0,C 180,E1 -9435.359,E2 -9435.359} C_VEL
LIN {X 0,Y 433.86,Z 651.692,A -85,B 0,C 180,E1 -9436.259,E2 -9436.259} C_VEL
LIN {X 0,Y 433.184,Z 662.737,A -85,B 0,C 180,E1 -9437.348,E2 -9437.348} C_VEL
LIN {X 0,Y 432.641,Z 672.313,A -85,B 0,C 180,E1 -9438.522,E2 -9438.522} C_VEL
LIN {X 0,Y 432.145,Z 680.13,A -85,B 0,C 180,E1 -9439.695,E2 -9439.695} C_VEL
LIN {X 0,Y 431.802,Z 687.741,A -85,B 0,C 180,E1 -9441.105,E2 -9441.105} C_VEL
LIN {X 0,Y 431.518,Z 693.848,A -85,B 0,C 180,E1 -9442.513,E2 -9442.513} C_VEL
LIN {X 0,Y 431.318,Z 698.842,A -85,B 0,C 180,E1 -9443.978,E2 -9443.978} C_VEL
LIN {X 0,Y 431.32,Z 702.35,A -85,B 0,C 180,E1 -9445.327,E2 -9445.327} C_VEL
LIN {X 0,Y 431.28,Z 704.245,A -85,B 0,C 180,E1 -9446.263,E2 -9446.263} C_VEL
LIN {X 0,Y 431.324,Z 705.678,A -85,B 0,C 180,E1 -9447.198,E2 -9447.198} C_VEL
LIN {X 0,Y 431.228,Z 707.302,A -85,B 0,C 180,E1 -9449.066,E2 -9449.066} C_VEL
LIN {X 0,Y 431.236,Z 707.523,A -85,B 0,C 180,E1 -9450,E2 -9450} C_VEL
LIN {X 0,Y 431.228,Z 707.301,A -85,B 0,C 180,E1 -9450.934,E2 -9450.934} C_VEL
LIN {X 0,Y 431.327,Z 705.677,A -85,B 0,C 180,E1 -9452.802,E2 -9452.802} C_VEL
LIN {X 0,Y 431.29,Z 704.242,A -85,B 0,C 180,E1 -9453.737,E2 -9453.737} C_VEL
LIN {X 0,Y 431.344,Z 701.26,A -85,B 0,C 180,E1 -9455.141,E2 -9455.141} C_VEL
LIN {X 0,Y 431.438,Z 697.209,A -85,B 0,C 180,E1 -9456.548,E2 -9456.548} C_VEL
LIN {X 0,Y 431.63,Z 690.957,A -85,B 0,C 180,E1 -9458.191,E2 -9458.191} C_VEL
LIN {X 0,Y 431.964,Z 684.136,A -85,B 0,C 180,E1 -9459.6,E2 -9459.6} C_VEL
LIN {X 0,Y 432.34,Z 677.151,A -85,B 0,C 180,E1 -9460.774,E2 -9460.774} C_VEL
LIN {X 0,Y 432.851,Z 668.708,A -85,B 0,C 180,E1 -9461.948,E2 -9461.948} C_VEL
LIN {X 0,Y 433.479,Z 658.249,A -85,B 0,C 180,E1 -9463.12,E2 -9463.12} C_VEL
LIN {X 0,Y 434.029,Z 647.874,A -85,B 0,C 180,E1 -9464.057,E2 -9464.057} C_VEL
LIN {X 0,Y 434.643,Z 636.422,A -85,B 0,C 180,E1 -9464.874,E2 -9464.874} C_VEL
LIN {X 0,Y 435.225,Z 624.509,A -85,B 0,C 180,E1 -9465.513,E2 -9465.513} C_VEL
LIN {X 0,Y 435.698,Z 611.605,A -85,B 0,C 180,E1 -9466.006,E2 -9466.006} C_VEL
LIN {X 0,Y 435.975,Z 599.395,A -85,B 0,C 180,E1 -9466.296,E2 -9466.296} C_VEL
LIN {X 0,Y 436.464,Z 567.902,A -85,B 0,C 180,E1 -9466.873,E2 -9466.873} C_VEL
LIN {X 0,Y 437.314,Z 516.692,A -85,B 0,C 180,E1 -9467.942,E2 -9467.942} C_VEL
LIN {X 0,Y 434.653,Z 492.692,A -85,B 0,C 180,E1 -9468.63,E2 -9468.63} C_VEL
LIN {X 0,Y 433.462,Z 484.933,A -85,B 0,C 180,E1 -9468.891,E2 -9468.891} C_VEL
LIN {X 0,Y 434.522,Z 465.333,A -85,B 0,C 180,E1 -9472.089,E2 -9472.089} C_VEL
LIN {X 0,Y 435.856,Z 444.875,A -85,B 0,C 180,E1 -9475.537,E2 -9475.537} C_VEL
LIN {X 0,Y 436.289,Z 437.603,A -85,B 0,C 180,E1 -9476.811,E2 -9476.811} C_VEL
LIN {X 0,Y 434.351,Z 427.593,A -85,B 0,C 180,E1 -9478.81,E2 -9478.81} C_VEL
LIN {X 0,Y 432.333,Z 419.637,A -85,B 0,C 180,E1 -9480.586,E2 -9480.586} C_VEL
LIN {X 0,Y 432.361,Z 419.63,A -85,B 0,C 180,E1 -9484.003,E2 -9484.003} C_VEL
LIN {X 0,Y 432.322,Z 419.635,A -85,B 0,C 180,E1 -9487.197,E2 -9487.197} C_VEL
LIN {X 0,Y 432.333,Z 419.632,A -85,B 0,C 180,E1 -9490.179,E2 -9490.179} C_VEL
LIN {X 0,Y 432.317,Z 419.636,A -85,B 0,C 180,E1 -9493.061,E2 -9493.061} C_VEL
LIN {X 0,Y 432.335,Z 419.633,A -85,B 0,C 180,E1 -9495.665,E2 -9495.665} C_VEL
LIN {X 0,Y 432.335,Z 419.629,A -85,B 0,C 180,E1 -9498.398,E2 -9498.398} C_VEL
LIN {X 0,Y 432.341,Z 419.63,A -85,B 0,C 180,E1 -9501.85,E2 -9501.85} C_VEL
LIN {X 0,Y 432.342,Z 419.63,A -85,B 0,C 180,E1 -9505.323,E2 -9505.323} C_VEL
LIN {X 0,Y 432.324,Z 419.634,A -85,B 0,C 180,E1 -9508.654,E2 -9508.654} C_VEL
LIN {X 0,Y 432.384,Z 419.626,A -85,B 0,C 180,E1 -9511.877,E2 -9511.877} C_VEL
LIN {X 0,Y 432.349,Z 419.634,A -85,B 0,C 180,E1 -9514.999,E2 -9514.999} C_VEL
LIN {X 0,Y 432.36,Z 419.631,A -85,B 0,C 180,E1 -9518.046,E2 -9518.046} C_VEL
LIN {X 0,Y 432.424,Z 419.778,A -85,B 0,C 180,E1 -9521.212,E2 -9521.212} C_VEL
LIN {X 0,Y 433.464,Z 422.578,A -85,B 0,C 180,E1 -9521.346,E2 -9521.346} C_VEL
LIN {X 0,Y 438.319,Z 434.047,A -85,B 0,C 180,E1 -9521.918,E2 -9521.918} C_VEL
LIN {X 0,Y 436.884,Z 502.51,A -85,B 0,C 180,E1 -9523.379,E2 -9523.379} C_VEL
LIN {X 0,Y 436.558,Z 523.599,A -85,B 0,C 180,E1 -9523.847,E2 -9523.847} C_VEL
LIN {X 0,Y 436.26,Z 535.842,A -85,B 0,C 180,E1 -9524.285,E2 -9524.285} C_VEL
LIN {X 0,Y 435.945,Z 547.502,A -85,B 0,C 180,E1 -9524.873,E2 -9524.873} C_VEL
LIN {X 0,Y 435.434,Z 559.479,A -85,B 0,C 180,E1 -9525.667,E2 -9525.667} C_VEL
LIN {X 0,Y 434.896,Z 570.164,A -85,B 0,C 180,E1 -9526.567,E2 -9526.567} C_VEL
LIN {X 0,Y 434.36,Z 580.229,A -85,B 0,C 180,E1 -9527.62,E2 -9527.62} C_VEL
LIN {X 0,Y 433.797,Z 589.257,A -85,B 0,C 180,E1 -9528.79,E2 -9528.79} C_VEL
LIN {X 0,Y 433.205,Z 598.025,A -85,B 0,C 180,E1 -9530.192,E2 -9530.192} C_VEL
LIN {X 0,Y 432.8,Z 605.01,A -85,B 0,C 180,E1 -9531.596,E2 -9531.596} C_VEL
LIN {X 0,Y 432.39,Z 611.02,A -85,B 0,C 180,E1 -9533.143,E2 -9533.143} C_VEL
LIN {X 0,Y 432.063,Z 614.852,A -85,B 0,C 180,E1 -9534.399,E2 -9534.399} C_VEL
LIN {X 0,Y 432.069,Z 617.091,A -85,B 0,C 180,E1 -9535.335,E2 -9535.335} C_VEL
LIN {X 0,Y 431.855,Z 618.917,A -85,B 0,C 180,E1 -9536.268,E2 -9536.268} C_VEL
LIN {X 0,Y 431.629,Z 620.262,A -85,B 0,C 180,E1 -9537.2,E2 -9537.2} C_VEL
LIN {X 0,Y 431.496,Z 621.179,A -85,B 0,C 180,E1 -9538.133,E2 -9538.133} C_VEL
LIN {X 0,Y 431.442,Z 621.689,A -85,B 0,C 180,E1 -9539.067,E2 -9539.067} C_VEL
LIN {X 0,Y 431.417,Z 621.773,A -85,B 0,C 180,E1 -9540,E2 -9540} C_VEL
LIN {X 0,Y 431.413,Z 621.415,A -85,B 0,C 180,E1 -9540.933,E2 -9540.933} C_VEL
LIN {X 0,Y 431.468,Z 620.654,A -85,B 0,C 180,E1 -9541.867,E2 -9541.867} C_VEL
LIN {X 0,Y 431.618,Z 619.483,A -85,B 0,C 180,E1 -9542.8,E2 -9542.8} C_VEL
LIN {X 0,Y 431.85,Z 616.888,A -85,B 0,C 180,E1 -9544.2,E2 -9544.2} C_VEL
LIN {X 0,Y 431.895,Z 613.284,A -85,B 0,C 180,E1 -9545.603,E2 -9545.603} C_VEL
LIN {X 0,Y 432.191,Z 607.453,A -85,B 0,C 180,E1 -9547.277,E2 -9547.277} C_VEL
LIN {X 0,Y 432.444,Z 601.344,A -85,B 0,C 180,E1 -9548.646,E2 -9548.646} C_VEL
LIN {X 0,Y 432.888,Z 593.546,A -85,B 0,C 180,E1 -9550.051,E2 -9550.051} C_VEL
LIN {X 0,Y 433.308,Z 585.554,A -85,B 0,C 180,E1 -9551.223,E2 -9551.223} C_VEL
LIN {X 0,Y 433.843,Z 574.689,A -85,B 0,C 180,E1 -9552.513,E2 -9552.513} C_VEL
LIN {X 0,Y 434.367,Z 564.612,A -85,B 0,C 180,E1 -9553.479,E2 -9553.479} C_VEL
LIN {X 0,Y 434.799,Z 552.706,A -85,B 0,C 180,E1 -9554.39,E2 -9554.39} C_VEL
LIN {X 0,Y 435.196,Z 539.706,A -85,B 0,C 180,E1 -9555.154,E2 -9555.154} C_VEL
LIN {X 0,Y 435.584,Z 526.456,A -85,B 0,C 180,E1 -9555.71,E2 -9555.71} C_VEL
LIN {X 0,Y 435.762,Z 512.301,A -85,B 0,C 180,E1 -9556.093,E2 -9556.093} C_VEL
LIN {X 0,Y 436.835,Z 432.841,A -85,B 0,C 180,E1 -9557.616,E2 -9557.616} C_VEL
LIN {X 0,Y 432.399,Z 419.627,A -85,B 0,C 180,E1 -9558.065,E2 -9558.065} C_VEL
LIN {X 0,Y 432.352,Z 419.633,A -85,B 0,C 180,E1 -9560.954,E2 -9560.954} C_VEL
LIN {X 0,Y 432.379,Z 419.621,A -85,B 0,C 180,E1 -9564.461,E2 -9564.461} C_VEL
LIN {X 0,Y 432.388,Z 419.625,A -85,B 0,C 180,E1 -9567.072,E2 -9567.072} C_VEL
LIN {X 0,Y 432.35,Z 419.627,A -85,B 0,C 180,E1 -9570.51,E2 -9570.51} C_VEL
LIN {X 0,Y 432.362,Z 419.612,A -85,B 0,C 180,E1 -9574.003,E2 -9574.003} C_VEL
LIN {X 0,Y 432.325,Z 419.637,A -85,B 0,C 180,E1 -9577.197,E2 -9577.197} C_VEL
LIN {X 0,Y 432.336,Z 419.621,A -85,B 0,C 180,E1 -9580.179,E2 -9580.179} C_VEL
LIN {X 0,Y 432.32,Z 419.638,A -85,B 0,C 180,E1 -9583.061,E2 -9583.061} C_VEL
LIN {X 0,Y 432.336,Z 419.619,A -85,B 0,C 180,E1 -9585.665,E2 -9585.665} C_VEL
LIN {X 0,Y 432.336,Z 419.633,A -85,B 0,C 180,E1 -9588.398,E2 -9588.398} C_VEL
LIN {X 0,Y 432.338,Z 419.63,A -85,B 0,C 180,E1 -9591.85,E2 -9591.85} C_VEL
LIN {X 0,Y 432.342,Z 419.628,A -85,B 0,C 180,E1 -9595.323,E2 -9595.323} C_VEL
LIN {X 0,Y 432.323,Z 419.637,A -85,B 0,C 180,E1 -9598.654,E2 -9598.654} C_VEL
LIN {X 0,Y 432.331,Z 419.638,A -85,B 0,C 180,E1 -9601.873,E2 -9601.873} C_VEL
LIN {X 0,Y 432.363,Z 419.739,A -85,B 0,C 180,E1 -9602.795,E2 -9602.795} C_VEL
LIN {X 0,Y 435.32,Z 433.872,A -85,B 0,C 180,E1 -9605.435,E2 -9605.435} C_VEL
LIN {X 0,Y 435.378,Z 440.956,A -85,B 0,C 180,E1 -9606.667,E2 -9606.667} C_VEL
LIN {X 0,Y 434.574,Z 459.967,A -85,B 0,C 180,E1 -9609.863,E2 -9609.863} C_VEL
LIN {X 0,Y 434.248,Z 471.255,A -85,B 0,C 180,E1 -9611.647,E2 -9611.647} C_VEL
LIN {X 0,Y 437.439,Z 489.979,A -85,B 0,C 180,E1 -9612.11,E2 -9612.11} C_VEL
LIN {X 0,Y 437.273,Z 504.461,A -85,B 0,C 180,E1 -9612.349,E2 -9612.349} C_VEL
LIN {X 0,Y 436.582,Z 510.311,A -85,B 0,C 180,E1 -9612.419,E2 -9612.419} C_VEL
LIN {X 0,Y 430.921,Z 529.34,A -85,B 0,C 180,E1 -9612.507,E2 -9612.507} C_VEL
LIN {X 0,Y 430.212,Z 535.192,A -85,B 0,C 180,E1 -9612.578,E2 -9612.578} C_VEL
LIN {X 0,Y 429.662,Z 582.245,A -85,B 0,C 180,E1 -9613.397,E2 -9613.397} C_VEL
LIN {X 0,Y 429.313,Z 595.219,A -85,B 0,C 180,E1 -9613.811,E2 -9613.811} C_VEL
LIN {X 0,Y 428.802,Z 607.085,A -85,B 0,C 180,E1 -9614.371,E2 -9614.371} C_VEL
LIN {X 0,Y 428.167,Z 619.212,A -85,B 0,C 180,E1 -9615.139,E2 -9615.139} C_VEL
LIN {X 0,Y 427.563,Z 630.506,A -85,B 0,C 180,E1 -9616.073,E2 -9616.073} C_VEL
LIN {X 0,Y 426.915,Z 640.951,A -85,B 0,C 180,E1 -9617.159,E2 -9617.159} C_VEL
LIN {X 0,Y 426.163,Z 650.246,A -85,B 0,C 180,E1 -9618.345,E2 -9618.345} C_VEL
LIN {X 0,Y 425.551,Z 659.206,A -85,B 0,C 180,E1 -9619.774,E2 -9619.774} C_VEL
LIN {X 0,Y 425.031,Z 666.397,A -85,B 0,C 180,E1 -9621.202,E2 -9621.202} C_VEL
LIN {X 0,Y 424.684,Z 671.277,A -85,B 0,C 180,E1 -9622.392,E2 -9622.392} C_VEL
LIN {X 0,Y 424.569,Z 675.421,A -85,B 0,C 180,E1 -9623.626,E2 -9623.626} C_VEL
LIN {X 0,Y 424.278,Z 679.61,A -85,B 0,C 180,E1 -9625.249,E2 -9625.249} C_VEL
LIN {X 0,Y 424.218,Z 681.47,A -85,B 0,C 180,E1 -9626.2,E2 -9626.2} C_VEL
LIN {X 0,Y 424.236,Z 682.89,A -85,B 0,C 180,E1 -9627.151,E2 -9627.151} C_VEL
LIN {X 0,Y 424.092,Z 684.504,A -85,B 0,C 180,E1 -9629.05,E2 -9629.05} C_VEL
LIN {X 0,Y 424.085,Z 684.74,A -85,B 0,C 180,E1 -9630,E2 -9630} C_VEL
LIN {X 0,Y 424.092,Z 684.55,A -85,B 0,C 180,E1 -9630.95,E2 -9630.95} C_VEL
LIN {X 0,Y 424.236,Z 682.997,A -85,B 0,C 180,E1 -9632.849,E2 -9632.849} C_VEL
LIN {X 0,Y 424.217,Z 681.636,A -85,B 0,C 180,E1 -9633.8,E2 -9633.8} C_VEL
LIN {X 0,Y 424.37,Z 678.768,A -85,B 0,C 180,E1 -9635.226,E2 -9635.226} C_VEL
LIN {X 0,Y 424.542,Z 674.872,A -85,B 0,C 180,E1 -9636.654,E2 -9636.654} C_VEL
LIN {X 0,Y 424.818,Z 669.825,A -85,B 0,C 180,E1 -9638.084,E2 -9638.084} C_VEL
LIN {X 0,Y 425.285,Z 663.458,A -85,B 0,C 180,E1 -9639.512,E2 -9639.512} C_VEL
LIN {X 0,Y 425.848,Z 655.549,A -85,B 0,C 180,E1 -9640.941,E2 -9640.941} C_VEL
LIN {X 0,Y 426.382,Z 647.47,A -85,B 0,C 180,E1 -9642.132,E2 -9642.132} C_VEL
LIN {X 0,Y 427.147,Z 637.541,A -85,B 0,C 180,E1 -9643.318,E2 -9643.318} C_VEL
LIN {X 0,Y 427.759,Z 626.385,A -85,B 0,C 180,E1 -9644.389,E2 -9644.389} C_VEL
LIN {X 0,Y 428.401,Z 615.465,A -85,B 0,C 180,E1 -9645.218,E2 -9645.218} C_VEL
LIN {X 0,Y 428.965,Z 604.409,A -85,B 0,C 180,E1 -9645.867,E2 -9645.867} C_VEL
LIN {X 0,Y 429.478,Z 591.282,A -85,B 0,C 180,E1 -9646.427,E2 -9646.427} C_VEL
LIN {X 0,Y 429.769,Z 579.794,A -85,B 0,C 180,E1 -9646.752,E2 -9646.752} C_VEL
LIN {X 0,Y 430.619,Z 489.974,A -85,B 0,C 180,E1 -9648.28,E2 -9648.28} C_VEL
LIN {X 0,Y 427.375,Z 471.361,A -85,B 0,C 180,E1 -9648.753,E2 -9648.753} C_VEL
LIN {X 0,Y 428.004,Z 453.405,A -85,B 0,C 180,E1 -9651.682,E2 -9651.682} C_VEL
LIN {X 0,Y 428.653,Z 437.255,A -85,B 0,C 180,E1 -9654.456,E2 -9654.456} C_VEL
LIN {X 0,Y 426.456,Z 425.72,A -85,B 0,C 180,E1 -9656.611,E2 -9656.611} C_VEL
LIN {X 0,Y 425.308,Z 420.511,A -85,B 0,C 180,E1 -9657.627,E2 -9657.627} C_VEL
LIN {X 0,Y 425.29,Z 420.51,A -85,B 0,C 180,E1 -9660.816,E2 -9660.816} C_VEL
LIN {X 0,Y 425.314,Z 420.508,A -85,B 0,C 180,E1 -9664.288,E2 -9664.288} C_VEL
LIN {X 0,Y 425.28,Z 420.51,A -85,B 0,C 180,E1 -9667.694,E2 -9667.694} C_VEL
LIN {X 0,Y 425.282,Z 420.504,A -85,B 0,C 180,E1 -9670.52,E2 -9670.52} C_VEL
LIN {X 0,Y 425.26,Z 420.509,A -85,B 0,C 180,E1 -9673.351,E2 -9673.351} C_VEL
LIN {X 0,Y 425.267,Z 420.515,A -85,B 0,C 180,E1 -9676.648,E2 -9676.648} C_VEL
LIN {X 0,Y 425.292,Z 420.506,A -85,B 0,C 180,E1 -9679.873,E2 -9679.873} C_VEL
LIN {X 0,Y 425.28,Z 420.507,A -85,B 0,C 180,E1 -9682.489,E2 -9682.489} C_VEL
LIN {X 0,Y 425.31,Z 420.503,A -85,B 0,C 180,E1 -9685.817,E2 -9685.817} C_VEL
LIN {X 0,Y 425.293,Z 420.508,A -85,B 0,C 180,E1 -9689.239,E2 -9689.239} C_VEL
LIN {X 0,Y 425.301,Z 420.509,A -85,B 0,C 180,E1 -9692.439,E2 -9692.439} C_VEL
LIN {X 0,Y 425.33,Z 420.616,A -85,B 0,C 180,E1 -9692.749,E2 -9692.749} C_VEL
LIN {X 0,Y 428.095,Z 434.32,A -85,B 0,C 180,E1 -9695.252,E2 -9695.252} C_VEL
LIN {X 0,Y 428.5,Z 439.015,A -85,B 0,C 180,E1 -9696.076,E2 -9696.076} C_VEL
LIN {X 0,Y 427.731,Z 456.504,A -85,B 0,C 180,E1 -9699.023,E2 -9699.023} C_VEL
LIN {X 0,Y 427.147,Z 471.954,A -85,B 0,C 180,E1 -9701.612,E2 -9701.612} C_VEL
LIN {X 0,Y 430.011,Z 490.767,A -85,B 0,C 180,E1 -9702.106,E2 -9702.106} C_VEL
LIN {X 0,Y 428.632,Z 581.859,A -85,B 0,C 180,E1 -9703.907,E2 -9703.907} C_VEL
LIN {X 0,Y 428.209,Z 595.714,A -85,B 0,C 180,E1 -9704.379,E2 -9704.379} C_VEL
LIN {X 0,Y 427.74,Z 608.312,A -85,B 0,C 180,E1 -9705.002,E2 -9705.002} C_VEL
LIN {X 0,Y 427.187,Z 620.414,A -85,B 0,C 180,E1 -9705.804,E2 -9705.804} C_VEL
LIN {X 0,Y 426.703,Z 632.026,A -85,B 0,C 180,E1 -9706.789,E2 -9706.789} C_VEL
LIN {X 0,Y 426.026,Z 643.157,A -85,B 0,C 180,E1 -9707.979,E2 -9707.979} C_VEL
LIN {X 0,Y 425.585,Z 651.355,A -85,B 0,C 180,E1 -9709.052,E2 -9709.052} C_VEL
LIN {X 0,Y 425.103,Z 660.247,A -85,B 0,C 180,E1 -9710.484,E2 -9710.484} C_VEL
LIN {X 0,Y 424.706,Z 667.407,A -85,B 0,C 180,E1 -9711.914,E2 -9711.914} C_VEL
LIN {X 0,Y 424.497,Z 673.277,A -85,B 0,C 180,E1 -9713.398,E2 -9713.398} C_VEL
LIN {X 0,Y 424.35,Z 677.522,A -85,B 0,C 180,E1 -9714.774,E2 -9714.774} C_VEL
LIN {X 0,Y 424.189,Z 680.831,A -85,B 0,C 180,E1 -9716.2,E2 -9716.2} C_VEL
LIN {X 0,Y 424.2,Z 682.462,A -85,B 0,C 180,E1 -9717.151,E2 -9717.151} C_VEL
LIN {X 0,Y 424.151,Z 683.67,A -85,B 0,C 180,E1 -9718.101,E2 -9718.101} C_VEL
LIN {X 0,Y 424.091,Z 684.409,A -85,B 0,C 180,E1 -9719.05,E2 -9719.05} C_VEL
LIN {X 0,Y 424.085,Z 684.747,A -85,B 0,C 180,E1 -9720,E2 -9720} C_VEL
LIN {X 0,Y 424.091,Z 684.673,A -85,B 0,C 180,E1 -9720.95,E2 -9720.95} C_VEL
LIN {X 0,Y 424.152,Z 684.131,A -85,B 0,C 180,E1 -9721.899,E2 -9721.899} C_VEL
LIN {X 0,Y 424.254,Z 683.185,A -85,B 0,C 180,E1 -9722.849,E2 -9722.849} C_VEL
LIN {X 0,Y 424.221,Z 681.824,A -85,B 0,C 180,E1 -9723.8,E2 -9723.8} C_VEL
LIN {X 0,Y 424.368,Z 678.898,A -85,B 0,C 180,E1 -9725.226,E2 -9725.226} C_VEL
LIN {X 0,Y 424.51,Z 674.886,A -85,B 0,C 180,E1 -9726.655,E2 -9726.655} C_VEL
LIN {X 0,Y 424.875,Z 668.694,A -85,B 0,C 180,E1 -9728.322,E2 -9728.322} C_VEL
LIN {X 0,Y 425.307,Z 661.872,A -85,B 0,C 180,E1 -9729.752,E2 -9729.752} C_VEL
LIN {X 0,Y 425.91,Z 653.315,A -85,B 0,C 180,E1 -9731.18,E2 -9731.18} C_VEL
LIN {X 0,Y 426.424,Z 644.589,A -85,B 0,C 180,E1 -9732.372,E2 -9732.372} C_VEL
LIN {X 0,Y 427.131,Z 634,A -85,B 0,C 180,E1 -9733.536,E2 -9733.536} C_VEL
LIN {X 0,Y 427.723,Z 623.029,A -85,B 0,C 180,E1 -9734.512,E2 -9734.512} C_VEL
LIN {X 0,Y 428.344,Z 611.101,A -85,B 0,C 180,E1 -9735.341,E2 -9735.341} C_VEL
LIN {X 0,Y 428.925,Z 598.945,A -85,B 0,C 180,E1 -9735.99,E2 -9735.99} C_VEL
LIN {X 0,Y 429.367,Z 585.623,A -85,B 0,C 180,E1 -9736.492,E2 -9736.492} C_VEL
LIN {X 0,Y 429.81,Z 567.635,A -85,B 0,C 180,E1 -9736.903,E2 -9736.903} C_VEL
LIN {X 0,Y 431.441,Z 490.44,A -85,B 0,C 180,E1 -9738.568,E2 -9738.568} C_VEL
LIN {X 0,Y 428.666,Z 475.122,A -85,B 0,C 180,E1 -9739.109,E2 -9739.109} C_VEL
LIN {X 0,Y 428.25,Z 473.007,A -85,B 0,C 180,E1 -9739.223,E2 -9739.223} C_VEL
LIN {X 0,Y 429.129,Z 454.044,A -85,B 0,C 180,E1 -9742.382,E2 -9742.382} C_VEL
LIN {X 0,Y 429.689,Z 440.389,A -85,B 0,C 180,E1 -9744.65,E2 -9744.65} C_VEL
LIN {X 0,Y 428.701,Z 433.778,A -85,B 0,C 180,E1 -9745.853,E2 -9745.853} C_VEL
LIN {X 0,Y 426.288,Z 423.972,A -85,B 0,C 180,E1 -9747.758,E2 -9747.758} C_VEL
LIN {X 0,Y 425.303,Z 420.511,A -85,B 0,C 180,E1 -9748.432,E2 -9748.432} C_VEL
LIN {X 0,Y 425.267,Z 420.515,A -85,B 0,C 180,E1 -9751.927,E2 -9751.927} C_VEL
LIN {X 0,Y 425.301,Z 420.509,A -85,B 0,C 180,E1 -9755.336,E2 -9755.336} C_VEL
LIN {X 0,Y 425.298,Z 420.51,A -85,B 0,C 180,E1 -9759.043,E2 -9759.043} C_VEL
LIN {X 0,Y 425.277,Z 420.512,A -85,B 0,C 180,E1 -9762.653,E2 -9762.653} C_VEL
LIN {X 0,Y 425.264,Z 420.512,A -85,B 0,C 180,E1 -9766.044,E2 -9766.044} C_VEL
LIN {X 0,Y 425.277,Z 420.511,A -85,B 0,C 180,E1 -9768.621,E2 -9768.621} C_VEL
LIN {X 0,Y 425.309,Z 420.505,A -85,B 0,C 180,E1 -9771.102,E2 -9771.102} C_VEL
LIN {X 0,Y 425.301,Z 420.507,A -85,B 0,C 180,E1 -9774.664,E2 -9774.664} C_VEL
LIN {X 0,Y 425.266,Z 420.511,A -85,B 0,C 180,E1 -9778.073,E2 -9778.073} C_VEL
LIN {X 0,Y 425.332,Z 420.678,A -85,B 0,C 180,E1 -9779.908,E2 -9779.908} C_VEL
LIN {X 0,Y 428.927,Z 437.491,A -85,B 0,C 180,E1 -9782.955,E2 -9782.955} C_VEL
LIN {X 0,Y 429.088,Z 442.205,A -85,B 0,C 180,E1 -9783.754,E2 -9783.754} C_VEL
LIN {X 0,Y 427.834,Z 463.991,A -85,B 0,C 180,E1 -9787.31,E2 -9787.31} C_VEL
LIN {X 0,Y 426.583,Z 487.31,A -85,B 0,C 180,E1 -9791.07,E2 -9791.07} C_VEL
LIN {X 0,Y 428.12,Z 499.973,A -85,B 0,C 180,E1 -9791.503,E2 -9791.503} C_VEL
LIN {X 0,Y 429.97,Z 518.168,A -85,B 0,C 180,E1 -9792.057,E2 -9792.057} C_VEL
LIN {X 0,Y 429.049,Z 602.475,A -85,B 0,C 180,E1 -9793.495,E2 -9793.495} C_VEL
LIN {X 0,Y 428.747,Z 615.195,A -85,B 0,C 180,E1 -9793.85,E2 -9793.85} C_VEL
LIN {X 0,Y 428.203,Z 628.034,A -85,B 0,C 180,E1 -9794.409,E2 -9794.409} C_VEL
LIN {X 0,Y 427.572,Z 639.858,A -85,B 0,C 180,E1 -9795.118,E2 -9795.118} C_VEL
LIN {X 0,Y 426.935,Z 651.551,A -85,B 0,C 180,E1 -9796.034,E2 -9796.034} C_VEL
LIN {X 0,Y 426.199,Z 662.559,A -85,B 0,C 180,E1 -9797.137,E2 -9797.137} C_VEL
LIN {X 0,Y 425.663,Z 672.133,A -85,B 0,C 180,E1 -9798.331,E2 -9798.331} C_VEL
LIN {X 0,Y 425.114,Z 679.947,A -85,B 0,C 180,E1 -9799.522,E2 -9799.522} C_VEL
LIN {X 0,Y 424.73,Z 687.555,A -85,B 0,C 180,E1 -9800.956,E2 -9800.956} C_VEL
LIN {X 0,Y 424.434,Z 693.661,A -85,B 0,C 180,E1 -9802.388,E2 -9802.388} C_VEL
LIN {X 0,Y 424.259,Z 698.068,A -85,B 0,C 180,E1 -9803.681,E2 -9803.681} C_VEL
LIN {X 0,Y 424.246,Z 702.162,A -85,B 0,C 180,E1 -9805.249,E2 -9805.249} C_VEL
LIN {X 0,Y 424.185,Z 704.057,A -85,B 0,C 180,E1 -9806.2,E2 -9806.2} C_VEL
LIN {X 0,Y 424.22,Z 705.491,A -85,B 0,C 180,E1 -9807.151,E2 -9807.151} C_VEL
LIN {X 0,Y 424.144,Z 707.13,A -85,B 0,C 180,E1 -9809.051,E2 -9809.051} C_VEL
LIN {X 0,Y 424.15,Z 707.334,A -85,B 0,C 180,E1 -9810,E2 -9810} C_VEL
LIN {X 0,Y 424.144,Z 707.112,A -85,B 0,C 180,E1 -9810.949,E2 -9810.949} C_VEL
LIN {X 0,Y 424.224,Z 705.487,A -85,B 0,C 180,E1 -9812.849,E2 -9812.849} C_VEL
LIN {X 0,Y 424.194,Z 704.053,A -85,B 0,C 180,E1 -9813.8,E2 -9813.8} C_VEL
LIN {X 0,Y 424.251,Z 701.071,A -85,B 0,C 180,E1 -9815.228,E2 -9815.228} C_VEL
LIN {X 0,Y 424.353,Z 697.02,A -85,B 0,C 180,E1 -9816.657,E2 -9816.657} C_VEL
LIN {X 0,Y 424.583,Z 690.769,A -85,B 0,C 180,E1 -9818.328,E2 -9818.328} C_VEL
LIN {X 0,Y 424.916,Z 683.948,A -85,B 0,C 180,E1 -9819.761,E2 -9819.761} C_VEL
LIN {X 0,Y 425.336,Z 676.965,A -85,B 0,C 180,E1 -9820.954,E2 -9820.954} C_VEL
LIN {X 0,Y 425.881,Z 668.524,A -85,B 0,C 180,E1 -9822.146,E2 -9822.146} C_VEL
LIN {X 0,Y 426.552,Z 658.068,A -85,B 0,C 180,E1 -9823.336,E2 -9823.336} C_VEL
LIN {X 0,Y 427.123,Z 647.696,A -85,B 0,C 180,E1 -9824.289,E2 -9824.289} C_VEL
LIN {X 0,Y 427.78,Z 636.251,A -85,B 0,C 180,E1 -9825.118,E2 -9825.118} C_VEL
LIN {X 0,Y 428.397,Z 624.349,A -85,B 0,C 180,E1 -9825.766,E2 -9825.766} C_VEL
LIN {X 0,Y 428.862,Z 611.463,A -85,B 0,C 180,E1 -9826.268,E2 -9826.268} C_VEL
LIN {X 0,Y 429.185,Z 599.306,A -85,B 0,C 180,E1 -9826.561,E2 -9826.561} C_VEL
LIN {X 0,Y 430.376,Z 535.747,A -85,B 0,C 180,E1 -9827.864,E2 -9827.864} C_VEL
LIN {X 0,Y 430.684,Z 517.621,A -85,B 0,C 180,E1 -9828.265,E2 -9828.265} C_VEL
LIN {X 0,Y 428.337,Z 495.101,A -85,B 0,C 180,E1 -9828.93,E2 -9828.93} C_VEL
LIN {X 0,Y 426.592,Z 483.896,A -85,B 0,C 180,E1 -9829.329,E2 -9829.329} C_VEL
LIN {X 0,Y 427.818,Z 463.968,A -85,B 0,C 180,E1 -9832.659,E2 -9832.659} C_VEL
LIN {X 0,Y 429.115,Z 445.309,A -85,B 0,C 180,E1 -9835.892,E2 -9835.892} C_VEL
LIN {X 0,Y 429.565,Z 440.532,A -85,B 0,C 180,E1 -9836.739,E2 -9836.739} C_VEL
LIN {X 0,Y 428.186,Z 432.172,A -85,B 0,C 180,E1 -9838.424,E2 -9838.424} C_VEL
LIN {X 0,Y 425.705,Z 422.175,A -85,B 0,C 180,E1 -9840.638,E2 -9840.638} C_VEL
LIN {X 0,Y 425.272,Z 420.517,A -85,B 0,C 180,E1 -9841.059,E2 -9841.059} C_VEL
LIN {X 0,Y 425.313,Z 420.507,A -85,B 0,C 180,E1 -9844.288,E2 -9844.288} C_VEL
LIN {X 0,Y 425.279,Z 420.513,A -85,B 0,C 180,E1 -9847.694,E2 -9847.694} C_VEL
LIN {X 0,Y 425.278,Z 420.511,A -85,B 0,C 180,E1 -9850.52,E2 -9850.52} C_VEL
LIN {X 0,Y 425.263,Z 420.513,A -85,B 0,C 180,E1 -9853.956,E2 -9853.956} C_VEL
LIN {X 0,Y 425.277,Z 420.514,A -85,B 0,C 180,E1 -9857.347,E2 -9857.347} C_VEL
LIN {X 0,Y 425.3,Z 420.509,A -85,B 0,C 180,E1 -9860.957,E2 -9860.957} C_VEL
LIN {X 0,Y 425.302,Z 420.507,A -85,B 0,C 180,E1 -9864.664,E2 -9864.664} C_VEL
LIN {X 0,Y 425.268,Z 420.512,A -85,B 0,C 180,E1 -9868.073,E2 -9868.073} C_VEL
LIN {X 0,Y 425.334,Z 420.505,A -85,B 0,C 180,E1 -9871.368,E2 -9871.368} C_VEL
LIN {X 0,Y 425.356,Z 420.503,A -85,B 0,C 180,E1 -9873.505,E2 -9873.505} C_VEL
LIN {X 0,Y 425.308,Z 420.513,A -85,B 0,C 180,E1 -9876.635,E2 -9876.635} C_VEL
LIN {X 0,Y 425.331,Z 420.507,A -85,B 0,C 180,E1 -9880.365,E2 -9880.365} C_VEL
LIN {X 0,Y 425.357,Z 420.594,A -85,B 0,C 180,E1 -9880.765,E2 -9880.765} C_VEL
LIN {X 0,Y 426.409,Z 423.463,A -85,B 0,C 180,E1 -9880.912,E2 -9880.912} C_VEL
LIN {X 0,Y 431.929,Z 436.05,A -85,B 0,C 180,E1 -9881.577,E2 -9881.577} C_VEL
LIN {X 0,Y 430.221,Z 504.412,A -85,B 0,C 180,E1 -9883.083,E2 -9883.083} C_VEL
